;FOLD SLIN P379 Vel=1 m/s CPDAT379 Tool[4]:Microflown3D Base[2]:straight_sol;%{PE}
;FOLD Parameters ;%{h}
;Params IlfProvider=kukaroboter.basistech.inlineforms.movement.spline; Kuka.IsGlobalPoint=False; Kuka.PointName=P379; Kuka.BlendingEnabled=False; Kuka.MoveDataName=CPDAT379; Kuka.VelocityPath=1.000; Kuka.VelocityFieldEnabled=True; Kuka.ColDetectFieldEnabled=True; Kuka.CurrentCDSetIndex=0; Kuka.MovementParameterFieldEnabled=True; IlfCommand=SLIN
;ENDFOLD
SLIN XP379 WITH $VEL = SVEL_CP(2.0, , LCPDAT379),$TOOL = STOOL2(FP379),$BASE = SBASE(FP379.BASE_NO),$IPO_MODE = SIPO_MODE(FP379.IPO_FRAME),$LOAD = SLOAD(FP379.TOOL_NO),$ACC = SACC_CP(LCPDAT379),$ORI_TYPE = SORI_TYP(LCPDAT379),$APO = SAPO(LCPDAT379),$JERK = SJERK(LCPDAT379),$COLLMON_TOL_PRO[1] = USE_CM_PRO_VALUES(0)
;ENDFOLD

;FOLD SLIN P380 Vel=1 m/s CPDAT380 Tool[4]:Microflown3D Base[2]:straight_sol;%{PE}
;FOLD Parameters ;%{h}
;Params IlfProvider=kukaroboter.basistech.inlineforms.movement.spline; Kuka.IsGlobalPoint=False; Kuka.PointName=P380; Kuka.BlendingEnabled=False; Kuka.MoveDataName=CPDAT380; Kuka.VelocityPath=1.000; Kuka.VelocityFieldEnabled=True; Kuka.ColDetectFieldEnabled=True; Kuka.CurrentCDSetIndex=0; Kuka.MovementParameterFieldEnabled=True; IlfCommand=SLIN
;ENDFOLD
SLIN XP380 WITH $VEL = SVEL_CP(2.0, , LCPDAT380),$TOOL = STOOL2(FP380),$BASE = SBASE(FP380.BASE_NO),$IPO_MODE = SIPO_MODE(FP380.IPO_FRAME),$LOAD = SLOAD(FP380.TOOL_NO),$ACC = SACC_CP(LCPDAT380),$ORI_TYPE = SORI_TYP(LCPDAT380),$APO = SAPO(LCPDAT380),$JERK = SJERK(LCPDAT380),$COLLMON_TOL_PRO[1] = USE_CM_PRO_VALUES(0)
;ENDFOLD

;FOLD SLIN P381 Vel=1 m/s CPDAT381 Tool[4]:Microflown3D Base[2]:straight_sol;%{PE}
;FOLD Parameters ;%{h}
;Params IlfProvider=kukaroboter.basistech.inlineforms.movement.spline; Kuka.IsGlobalPoint=False; Kuka.PointName=P381; Kuka.BlendingEnabled=False; Kuka.MoveDataName=CPDAT381; Kuka.VelocityPath=1.000; Kuka.VelocityFieldEnabled=True; Kuka.ColDetectFieldEnabled=True; Kuka.CurrentCDSetIndex=0; Kuka.MovementParameterFieldEnabled=True; IlfCommand=SLIN
;ENDFOLD
SLIN XP381 WITH $VEL = SVEL_CP(2.0, , LCPDAT381),$TOOL = STOOL2(FP381),$BASE = SBASE(FP381.BASE_NO),$IPO_MODE = SIPO_MODE(FP381.IPO_FRAME),$LOAD = SLOAD(FP381.TOOL_NO),$ACC = SACC_CP(LCPDAT381),$ORI_TYPE = SORI_TYP(LCPDAT381),$APO = SAPO(LCPDAT381),$JERK = SJERK(LCPDAT381),$COLLMON_TOL_PRO[1] = USE_CM_PRO_VALUES(0)
;ENDFOLD

;FOLD SLIN P382 Vel=1 m/s CPDAT382 Tool[4]:Microflown3D Base[2]:straight_sol;%{PE}
;FOLD Parameters ;%{h}
;Params IlfProvider=kukaroboter.basistech.inlineforms.movement.spline; Kuka.IsGlobalPoint=False; Kuka.PointName=P382; Kuka.BlendingEnabled=False; Kuka.MoveDataName=CPDAT382; Kuka.VelocityPath=1.000; Kuka.VelocityFieldEnabled=True; Kuka.ColDetectFieldEnabled=True; Kuka.CurrentCDSetIndex=0; Kuka.MovementParameterFieldEnabled=True; IlfCommand=SLIN
;ENDFOLD
SLIN XP382 WITH $VEL = SVEL_CP(2.0, , LCPDAT382),$TOOL = STOOL2(FP382),$BASE = SBASE(FP382.BASE_NO),$IPO_MODE = SIPO_MODE(FP382.IPO_FRAME),$LOAD = SLOAD(FP382.TOOL_NO),$ACC = SACC_CP(LCPDAT382),$ORI_TYPE = SORI_TYP(LCPDAT382),$APO = SAPO(LCPDAT382),$JERK = SJERK(LCPDAT382),$COLLMON_TOL_PRO[1] = USE_CM_PRO_VALUES(0)
;ENDFOLD

;FOLD SLIN P383 Vel=1 m/s CPDAT383 Tool[4]:Microflown3D Base[2]:straight_sol;%{PE}
;FOLD Parameters ;%{h}
;Params IlfProvider=kukaroboter.basistech.inlineforms.movement.spline; Kuka.IsGlobalPoint=False; Kuka.PointName=P383; Kuka.BlendingEnabled=False; Kuka.MoveDataName=CPDAT383; Kuka.VelocityPath=1.000; Kuka.VelocityFieldEnabled=True; Kuka.ColDetectFieldEnabled=True; Kuka.CurrentCDSetIndex=0; Kuka.MovementParameterFieldEnabled=True; IlfCommand=SLIN
;ENDFOLD
SLIN XP383 WITH $VEL = SVEL_CP(2.0, , LCPDAT383),$TOOL = STOOL2(FP383),$BASE = SBASE(FP383.BASE_NO),$IPO_MODE = SIPO_MODE(FP383.IPO_FRAME),$LOAD = SLOAD(FP383.TOOL_NO),$ACC = SACC_CP(LCPDAT383),$ORI_TYPE = SORI_TYP(LCPDAT383),$APO = SAPO(LCPDAT383),$JERK = SJERK(LCPDAT383),$COLLMON_TOL_PRO[1] = USE_CM_PRO_VALUES(0)
;ENDFOLD

;FOLD SLIN P384 Vel=1 m/s CPDAT384 Tool[4]:Microflown3D Base[2]:straight_sol;%{PE}
;FOLD Parameters ;%{h}
;Params IlfProvider=kukaroboter.basistech.inlineforms.movement.spline; Kuka.IsGlobalPoint=False; Kuka.PointName=P384; Kuka.BlendingEnabled=False; Kuka.MoveDataName=CPDAT384; Kuka.VelocityPath=1.000; Kuka.VelocityFieldEnabled=True; Kuka.ColDetectFieldEnabled=True; Kuka.CurrentCDSetIndex=0; Kuka.MovementParameterFieldEnabled=True; IlfCommand=SLIN
;ENDFOLD
SLIN XP384 WITH $VEL = SVEL_CP(2.0, , LCPDAT384),$TOOL = STOOL2(FP384),$BASE = SBASE(FP384.BASE_NO),$IPO_MODE = SIPO_MODE(FP384.IPO_FRAME),$LOAD = SLOAD(FP384.TOOL_NO),$ACC = SACC_CP(LCPDAT384),$ORI_TYPE = SORI_TYP(LCPDAT384),$APO = SAPO(LCPDAT384),$JERK = SJERK(LCPDAT384),$COLLMON_TOL_PRO[1] = USE_CM_PRO_VALUES(0)
;ENDFOLD

;FOLD SLIN P385 Vel=1 m/s CPDAT385 Tool[4]:Microflown3D Base[2]:straight_sol;%{PE}
;FOLD Parameters ;%{h}
;Params IlfProvider=kukaroboter.basistech.inlineforms.movement.spline; Kuka.IsGlobalPoint=False; Kuka.PointName=P385; Kuka.BlendingEnabled=False; Kuka.MoveDataName=CPDAT385; Kuka.VelocityPath=1.000; Kuka.VelocityFieldEnabled=True; Kuka.ColDetectFieldEnabled=True; Kuka.CurrentCDSetIndex=0; Kuka.MovementParameterFieldEnabled=True; IlfCommand=SLIN
;ENDFOLD
SLIN XP385 WITH $VEL = SVEL_CP(2.0, , LCPDAT385),$TOOL = STOOL2(FP385),$BASE = SBASE(FP385.BASE_NO),$IPO_MODE = SIPO_MODE(FP385.IPO_FRAME),$LOAD = SLOAD(FP385.TOOL_NO),$ACC = SACC_CP(LCPDAT385),$ORI_TYPE = SORI_TYP(LCPDAT385),$APO = SAPO(LCPDAT385),$JERK = SJERK(LCPDAT385),$COLLMON_TOL_PRO[1] = USE_CM_PRO_VALUES(0)
;ENDFOLD

;FOLD SLIN P386 Vel=1 m/s CPDAT386 Tool[4]:Microflown3D Base[2]:straight_sol;%{PE}
;FOLD Parameters ;%{h}
;Params IlfProvider=kukaroboter.basistech.inlineforms.movement.spline; Kuka.IsGlobalPoint=False; Kuka.PointName=P386; Kuka.BlendingEnabled=False; Kuka.MoveDataName=CPDAT386; Kuka.VelocityPath=1.000; Kuka.VelocityFieldEnabled=True; Kuka.ColDetectFieldEnabled=True; Kuka.CurrentCDSetIndex=0; Kuka.MovementParameterFieldEnabled=True; IlfCommand=SLIN
;ENDFOLD
SLIN XP386 WITH $VEL = SVEL_CP(2.0, , LCPDAT386),$TOOL = STOOL2(FP386),$BASE = SBASE(FP386.BASE_NO),$IPO_MODE = SIPO_MODE(FP386.IPO_FRAME),$LOAD = SLOAD(FP386.TOOL_NO),$ACC = SACC_CP(LCPDAT386),$ORI_TYPE = SORI_TYP(LCPDAT386),$APO = SAPO(LCPDAT386),$JERK = SJERK(LCPDAT386),$COLLMON_TOL_PRO[1] = USE_CM_PRO_VALUES(0)
;ENDFOLD

;FOLD SLIN P387 Vel=1 m/s CPDAT387 Tool[4]:Microflown3D Base[2]:straight_sol;%{PE}
;FOLD Parameters ;%{h}
;Params IlfProvider=kukaroboter.basistech.inlineforms.movement.spline; Kuka.IsGlobalPoint=False; Kuka.PointName=P387; Kuka.BlendingEnabled=False; Kuka.MoveDataName=CPDAT387; Kuka.VelocityPath=1.000; Kuka.VelocityFieldEnabled=True; Kuka.ColDetectFieldEnabled=True; Kuka.CurrentCDSetIndex=0; Kuka.MovementParameterFieldEnabled=True; IlfCommand=SLIN
;ENDFOLD
SLIN XP387 WITH $VEL = SVEL_CP(2.0, , LCPDAT387),$TOOL = STOOL2(FP387),$BASE = SBASE(FP387.BASE_NO),$IPO_MODE = SIPO_MODE(FP387.IPO_FRAME),$LOAD = SLOAD(FP387.TOOL_NO),$ACC = SACC_CP(LCPDAT387),$ORI_TYPE = SORI_TYP(LCPDAT387),$APO = SAPO(LCPDAT387),$JERK = SJERK(LCPDAT387),$COLLMON_TOL_PRO[1] = USE_CM_PRO_VALUES(0)
;ENDFOLD

;FOLD SLIN P388 Vel=1 m/s CPDAT388 Tool[4]:Microflown3D Base[2]:straight_sol;%{PE}
;FOLD Parameters ;%{h}
;Params IlfProvider=kukaroboter.basistech.inlineforms.movement.spline; Kuka.IsGlobalPoint=False; Kuka.PointName=P388; Kuka.BlendingEnabled=False; Kuka.MoveDataName=CPDAT388; Kuka.VelocityPath=1.000; Kuka.VelocityFieldEnabled=True; Kuka.ColDetectFieldEnabled=True; Kuka.CurrentCDSetIndex=0; Kuka.MovementParameterFieldEnabled=True; IlfCommand=SLIN
;ENDFOLD
SLIN XP388 WITH $VEL = SVEL_CP(2.0, , LCPDAT388),$TOOL = STOOL2(FP388),$BASE = SBASE(FP388.BASE_NO),$IPO_MODE = SIPO_MODE(FP388.IPO_FRAME),$LOAD = SLOAD(FP388.TOOL_NO),$ACC = SACC_CP(LCPDAT388),$ORI_TYPE = SORI_TYP(LCPDAT388),$APO = SAPO(LCPDAT388),$JERK = SJERK(LCPDAT388),$COLLMON_TOL_PRO[1] = USE_CM_PRO_VALUES(0)
;ENDFOLD

;FOLD SLIN P389 Vel=1 m/s CPDAT389 Tool[4]:Microflown3D Base[2]:straight_sol;%{PE}
;FOLD Parameters ;%{h}
;Params IlfProvider=kukaroboter.basistech.inlineforms.movement.spline; Kuka.IsGlobalPoint=False; Kuka.PointName=P389; Kuka.BlendingEnabled=False; Kuka.MoveDataName=CPDAT389; Kuka.VelocityPath=1.000; Kuka.VelocityFieldEnabled=True; Kuka.ColDetectFieldEnabled=True; Kuka.CurrentCDSetIndex=0; Kuka.MovementParameterFieldEnabled=True; IlfCommand=SLIN
;ENDFOLD
SLIN XP389 WITH $VEL = SVEL_CP(2.0, , LCPDAT389),$TOOL = STOOL2(FP389),$BASE = SBASE(FP389.BASE_NO),$IPO_MODE = SIPO_MODE(FP389.IPO_FRAME),$LOAD = SLOAD(FP389.TOOL_NO),$ACC = SACC_CP(LCPDAT389),$ORI_TYPE = SORI_TYP(LCPDAT389),$APO = SAPO(LCPDAT389),$JERK = SJERK(LCPDAT389),$COLLMON_TOL_PRO[1] = USE_CM_PRO_VALUES(0)
;ENDFOLD

;FOLD SLIN P390 Vel=1 m/s CPDAT390 Tool[4]:Microflown3D Base[2]:straight_sol;%{PE}
;FOLD Parameters ;%{h}
;Params IlfProvider=kukaroboter.basistech.inlineforms.movement.spline; Kuka.IsGlobalPoint=False; Kuka.PointName=P390; Kuka.BlendingEnabled=False; Kuka.MoveDataName=CPDAT390; Kuka.VelocityPath=1.000; Kuka.VelocityFieldEnabled=True; Kuka.ColDetectFieldEnabled=True; Kuka.CurrentCDSetIndex=0; Kuka.MovementParameterFieldEnabled=True; IlfCommand=SLIN
;ENDFOLD
SLIN XP390 WITH $VEL = SVEL_CP(2.0, , LCPDAT390),$TOOL = STOOL2(FP390),$BASE = SBASE(FP390.BASE_NO),$IPO_MODE = SIPO_MODE(FP390.IPO_FRAME),$LOAD = SLOAD(FP390.TOOL_NO),$ACC = SACC_CP(LCPDAT390),$ORI_TYPE = SORI_TYP(LCPDAT390),$APO = SAPO(LCPDAT390),$JERK = SJERK(LCPDAT390),$COLLMON_TOL_PRO[1] = USE_CM_PRO_VALUES(0)
;ENDFOLD

;FOLD SLIN P391 Vel=1 m/s CPDAT391 Tool[4]:Microflown3D Base[2]:straight_sol;%{PE}
;FOLD Parameters ;%{h}
;Params IlfProvider=kukaroboter.basistech.inlineforms.movement.spline; Kuka.IsGlobalPoint=False; Kuka.PointName=P391; Kuka.BlendingEnabled=False; Kuka.MoveDataName=CPDAT391; Kuka.VelocityPath=1.000; Kuka.VelocityFieldEnabled=True; Kuka.ColDetectFieldEnabled=True; Kuka.CurrentCDSetIndex=0; Kuka.MovementParameterFieldEnabled=True; IlfCommand=SLIN
;ENDFOLD
SLIN XP391 WITH $VEL = SVEL_CP(2.0, , LCPDAT391),$TOOL = STOOL2(FP391),$BASE = SBASE(FP391.BASE_NO),$IPO_MODE = SIPO_MODE(FP391.IPO_FRAME),$LOAD = SLOAD(FP391.TOOL_NO),$ACC = SACC_CP(LCPDAT391),$ORI_TYPE = SORI_TYP(LCPDAT391),$APO = SAPO(LCPDAT391),$JERK = SJERK(LCPDAT391),$COLLMON_TOL_PRO[1] = USE_CM_PRO_VALUES(0)
;ENDFOLD

;FOLD SLIN P392 Vel=1 m/s CPDAT392 Tool[4]:Microflown3D Base[2]:straight_sol;%{PE}
;FOLD Parameters ;%{h}
;Params IlfProvider=kukaroboter.basistech.inlineforms.movement.spline; Kuka.IsGlobalPoint=False; Kuka.PointName=P392; Kuka.BlendingEnabled=False; Kuka.MoveDataName=CPDAT392; Kuka.VelocityPath=1.000; Kuka.VelocityFieldEnabled=True; Kuka.ColDetectFieldEnabled=True; Kuka.CurrentCDSetIndex=0; Kuka.MovementParameterFieldEnabled=True; IlfCommand=SLIN
;ENDFOLD
SLIN XP392 WITH $VEL = SVEL_CP(2.0, , LCPDAT392),$TOOL = STOOL2(FP392),$BASE = SBASE(FP392.BASE_NO),$IPO_MODE = SIPO_MODE(FP392.IPO_FRAME),$LOAD = SLOAD(FP392.TOOL_NO),$ACC = SACC_CP(LCPDAT392),$ORI_TYPE = SORI_TYP(LCPDAT392),$APO = SAPO(LCPDAT392),$JERK = SJERK(LCPDAT392),$COLLMON_TOL_PRO[1] = USE_CM_PRO_VALUES(0)
;ENDFOLD

;FOLD SLIN P393 Vel=1 m/s CPDAT393 Tool[4]:Microflown3D Base[2]:straight_sol;%{PE}
;FOLD Parameters ;%{h}
;Params IlfProvider=kukaroboter.basistech.inlineforms.movement.spline; Kuka.IsGlobalPoint=False; Kuka.PointName=P393; Kuka.BlendingEnabled=False; Kuka.MoveDataName=CPDAT393; Kuka.VelocityPath=1.000; Kuka.VelocityFieldEnabled=True; Kuka.ColDetectFieldEnabled=True; Kuka.CurrentCDSetIndex=0; Kuka.MovementParameterFieldEnabled=True; IlfCommand=SLIN
;ENDFOLD
SLIN XP393 WITH $VEL = SVEL_CP(2.0, , LCPDAT393),$TOOL = STOOL2(FP393),$BASE = SBASE(FP393.BASE_NO),$IPO_MODE = SIPO_MODE(FP393.IPO_FRAME),$LOAD = SLOAD(FP393.TOOL_NO),$ACC = SACC_CP(LCPDAT393),$ORI_TYPE = SORI_TYP(LCPDAT393),$APO = SAPO(LCPDAT393),$JERK = SJERK(LCPDAT393),$COLLMON_TOL_PRO[1] = USE_CM_PRO_VALUES(0)
;ENDFOLD

;FOLD SLIN P394 Vel=1 m/s CPDAT394 Tool[4]:Microflown3D Base[2]:straight_sol;%{PE}
;FOLD Parameters ;%{h}
;Params IlfProvider=kukaroboter.basistech.inlineforms.movement.spline; Kuka.IsGlobalPoint=False; Kuka.PointName=P394; Kuka.BlendingEnabled=False; Kuka.MoveDataName=CPDAT394; Kuka.VelocityPath=1.000; Kuka.VelocityFieldEnabled=True; Kuka.ColDetectFieldEnabled=True; Kuka.CurrentCDSetIndex=0; Kuka.MovementParameterFieldEnabled=True; IlfCommand=SLIN
;ENDFOLD
SLIN XP394 WITH $VEL = SVEL_CP(2.0, , LCPDAT394),$TOOL = STOOL2(FP394),$BASE = SBASE(FP394.BASE_NO),$IPO_MODE = SIPO_MODE(FP394.IPO_FRAME),$LOAD = SLOAD(FP394.TOOL_NO),$ACC = SACC_CP(LCPDAT394),$ORI_TYPE = SORI_TYP(LCPDAT394),$APO = SAPO(LCPDAT394),$JERK = SJERK(LCPDAT394),$COLLMON_TOL_PRO[1] = USE_CM_PRO_VALUES(0)
;ENDFOLD

;FOLD SLIN P395 Vel=1 m/s CPDAT395 Tool[4]:Microflown3D Base[2]:straight_sol;%{PE}
;FOLD Parameters ;%{h}
;Params IlfProvider=kukaroboter.basistech.inlineforms.movement.spline; Kuka.IsGlobalPoint=False; Kuka.PointName=P395; Kuka.BlendingEnabled=False; Kuka.MoveDataName=CPDAT395; Kuka.VelocityPath=1.000; Kuka.VelocityFieldEnabled=True; Kuka.ColDetectFieldEnabled=True; Kuka.CurrentCDSetIndex=0; Kuka.MovementParameterFieldEnabled=True; IlfCommand=SLIN
;ENDFOLD
SLIN XP395 WITH $VEL = SVEL_CP(2.0, , LCPDAT395),$TOOL = STOOL2(FP395),$BASE = SBASE(FP395.BASE_NO),$IPO_MODE = SIPO_MODE(FP395.IPO_FRAME),$LOAD = SLOAD(FP395.TOOL_NO),$ACC = SACC_CP(LCPDAT395),$ORI_TYPE = SORI_TYP(LCPDAT395),$APO = SAPO(LCPDAT395),$JERK = SJERK(LCPDAT395),$COLLMON_TOL_PRO[1] = USE_CM_PRO_VALUES(0)
;ENDFOLD

;FOLD SLIN P396 Vel=1 m/s CPDAT396 Tool[4]:Microflown3D Base[2]:straight_sol;%{PE}
;FOLD Parameters ;%{h}
;Params IlfProvider=kukaroboter.basistech.inlineforms.movement.spline; Kuka.IsGlobalPoint=False; Kuka.PointName=P396; Kuka.BlendingEnabled=False; Kuka.MoveDataName=CPDAT396; Kuka.VelocityPath=1.000; Kuka.VelocityFieldEnabled=True; Kuka.ColDetectFieldEnabled=True; Kuka.CurrentCDSetIndex=0; Kuka.MovementParameterFieldEnabled=True; IlfCommand=SLIN
;ENDFOLD
SLIN XP396 WITH $VEL = SVEL_CP(2.0, , LCPDAT396),$TOOL = STOOL2(FP396),$BASE = SBASE(FP396.BASE_NO),$IPO_MODE = SIPO_MODE(FP396.IPO_FRAME),$LOAD = SLOAD(FP396.TOOL_NO),$ACC = SACC_CP(LCPDAT396),$ORI_TYPE = SORI_TYP(LCPDAT396),$APO = SAPO(LCPDAT396),$JERK = SJERK(LCPDAT396),$COLLMON_TOL_PRO[1] = USE_CM_PRO_VALUES(0)
;ENDFOLD

;FOLD SLIN P397 Vel=1 m/s CPDAT397 Tool[4]:Microflown3D Base[2]:straight_sol;%{PE}
;FOLD Parameters ;%{h}
;Params IlfProvider=kukaroboter.basistech.inlineforms.movement.spline; Kuka.IsGlobalPoint=False; Kuka.PointName=P397; Kuka.BlendingEnabled=False; Kuka.MoveDataName=CPDAT397; Kuka.VelocityPath=1.000; Kuka.VelocityFieldEnabled=True; Kuka.ColDetectFieldEnabled=True; Kuka.CurrentCDSetIndex=0; Kuka.MovementParameterFieldEnabled=True; IlfCommand=SLIN
;ENDFOLD
SLIN XP397 WITH $VEL = SVEL_CP(2.0, , LCPDAT397),$TOOL = STOOL2(FP397),$BASE = SBASE(FP397.BASE_NO),$IPO_MODE = SIPO_MODE(FP397.IPO_FRAME),$LOAD = SLOAD(FP397.TOOL_NO),$ACC = SACC_CP(LCPDAT397),$ORI_TYPE = SORI_TYP(LCPDAT397),$APO = SAPO(LCPDAT397),$JERK = SJERK(LCPDAT397),$COLLMON_TOL_PRO[1] = USE_CM_PRO_VALUES(0)
;ENDFOLD

;FOLD SLIN P398 Vel=1 m/s CPDAT398 Tool[4]:Microflown3D Base[2]:straight_sol;%{PE}
;FOLD Parameters ;%{h}
;Params IlfProvider=kukaroboter.basistech.inlineforms.movement.spline; Kuka.IsGlobalPoint=False; Kuka.PointName=P398; Kuka.BlendingEnabled=False; Kuka.MoveDataName=CPDAT398; Kuka.VelocityPath=1.000; Kuka.VelocityFieldEnabled=True; Kuka.ColDetectFieldEnabled=True; Kuka.CurrentCDSetIndex=0; Kuka.MovementParameterFieldEnabled=True; IlfCommand=SLIN
;ENDFOLD
SLIN XP398 WITH $VEL = SVEL_CP(2.0, , LCPDAT398),$TOOL = STOOL2(FP398),$BASE = SBASE(FP398.BASE_NO),$IPO_MODE = SIPO_MODE(FP398.IPO_FRAME),$LOAD = SLOAD(FP398.TOOL_NO),$ACC = SACC_CP(LCPDAT398),$ORI_TYPE = SORI_TYP(LCPDAT398),$APO = SAPO(LCPDAT398),$JERK = SJERK(LCPDAT398),$COLLMON_TOL_PRO[1] = USE_CM_PRO_VALUES(0)
;ENDFOLD

;FOLD SLIN P399 Vel=1 m/s CPDAT399 Tool[4]:Microflown3D Base[2]:straight_sol;%{PE}
;FOLD Parameters ;%{h}
;Params IlfProvider=kukaroboter.basistech.inlineforms.movement.spline; Kuka.IsGlobalPoint=False; Kuka.PointName=P399; Kuka.BlendingEnabled=False; Kuka.MoveDataName=CPDAT399; Kuka.VelocityPath=1.000; Kuka.VelocityFieldEnabled=True; Kuka.ColDetectFieldEnabled=True; Kuka.CurrentCDSetIndex=0; Kuka.MovementParameterFieldEnabled=True; IlfCommand=SLIN
;ENDFOLD
SLIN XP399 WITH $VEL = SVEL_CP(2.0, , LCPDAT399),$TOOL = STOOL2(FP399),$BASE = SBASE(FP399.BASE_NO),$IPO_MODE = SIPO_MODE(FP399.IPO_FRAME),$LOAD = SLOAD(FP399.TOOL_NO),$ACC = SACC_CP(LCPDAT399),$ORI_TYPE = SORI_TYP(LCPDAT399),$APO = SAPO(LCPDAT399),$JERK = SJERK(LCPDAT399),$COLLMON_TOL_PRO[1] = USE_CM_PRO_VALUES(0)
;ENDFOLD

;FOLD SLIN P400 Vel=1 m/s CPDAT400 Tool[4]:Microflown3D Base[2]:straight_sol;%{PE}
;FOLD Parameters ;%{h}
;Params IlfProvider=kukaroboter.basistech.inlineforms.movement.spline; Kuka.IsGlobalPoint=False; Kuka.PointName=P400; Kuka.BlendingEnabled=False; Kuka.MoveDataName=CPDAT400; Kuka.VelocityPath=1.000; Kuka.VelocityFieldEnabled=True; Kuka.ColDetectFieldEnabled=True; Kuka.CurrentCDSetIndex=0; Kuka.MovementParameterFieldEnabled=True; IlfCommand=SLIN
;ENDFOLD
SLIN XP400 WITH $VEL = SVEL_CP(2.0, , LCPDAT400),$TOOL = STOOL2(FP400),$BASE = SBASE(FP400.BASE_NO),$IPO_MODE = SIPO_MODE(FP400.IPO_FRAME),$LOAD = SLOAD(FP400.TOOL_NO),$ACC = SACC_CP(LCPDAT400),$ORI_TYPE = SORI_TYP(LCPDAT400),$APO = SAPO(LCPDAT400),$JERK = SJERK(LCPDAT400),$COLLMON_TOL_PRO[1] = USE_CM_PRO_VALUES(0)
;ENDFOLD

;FOLD SLIN P401 Vel=1 m/s CPDAT401 Tool[4]:Microflown3D Base[2]:straight_sol;%{PE}
;FOLD Parameters ;%{h}
;Params IlfProvider=kukaroboter.basistech.inlineforms.movement.spline; Kuka.IsGlobalPoint=False; Kuka.PointName=P401; Kuka.BlendingEnabled=False; Kuka.MoveDataName=CPDAT401; Kuka.VelocityPath=1.000; Kuka.VelocityFieldEnabled=True; Kuka.ColDetectFieldEnabled=True; Kuka.CurrentCDSetIndex=0; Kuka.MovementParameterFieldEnabled=True; IlfCommand=SLIN
;ENDFOLD
SLIN XP401 WITH $VEL = SVEL_CP(2.0, , LCPDAT401),$TOOL = STOOL2(FP401),$BASE = SBASE(FP401.BASE_NO),$IPO_MODE = SIPO_MODE(FP401.IPO_FRAME),$LOAD = SLOAD(FP401.TOOL_NO),$ACC = SACC_CP(LCPDAT401),$ORI_TYPE = SORI_TYP(LCPDAT401),$APO = SAPO(LCPDAT401),$JERK = SJERK(LCPDAT401),$COLLMON_TOL_PRO[1] = USE_CM_PRO_VALUES(0)
;ENDFOLD

;FOLD SLIN P402 Vel=1 m/s CPDAT402 Tool[4]:Microflown3D Base[2]:straight_sol;%{PE}
;FOLD Parameters ;%{h}
;Params IlfProvider=kukaroboter.basistech.inlineforms.movement.spline; Kuka.IsGlobalPoint=False; Kuka.PointName=P402; Kuka.BlendingEnabled=False; Kuka.MoveDataName=CPDAT402; Kuka.VelocityPath=1.000; Kuka.VelocityFieldEnabled=True; Kuka.ColDetectFieldEnabled=True; Kuka.CurrentCDSetIndex=0; Kuka.MovementParameterFieldEnabled=True; IlfCommand=SLIN
;ENDFOLD
SLIN XP402 WITH $VEL = SVEL_CP(2.0, , LCPDAT402),$TOOL = STOOL2(FP402),$BASE = SBASE(FP402.BASE_NO),$IPO_MODE = SIPO_MODE(FP402.IPO_FRAME),$LOAD = SLOAD(FP402.TOOL_NO),$ACC = SACC_CP(LCPDAT402),$ORI_TYPE = SORI_TYP(LCPDAT402),$APO = SAPO(LCPDAT402),$JERK = SJERK(LCPDAT402),$COLLMON_TOL_PRO[1] = USE_CM_PRO_VALUES(0)
;ENDFOLD

;FOLD SLIN P403 Vel=1 m/s CPDAT403 Tool[4]:Microflown3D Base[2]:straight_sol;%{PE}
;FOLD Parameters ;%{h}
;Params IlfProvider=kukaroboter.basistech.inlineforms.movement.spline; Kuka.IsGlobalPoint=False; Kuka.PointName=P403; Kuka.BlendingEnabled=False; Kuka.MoveDataName=CPDAT403; Kuka.VelocityPath=1.000; Kuka.VelocityFieldEnabled=True; Kuka.ColDetectFieldEnabled=True; Kuka.CurrentCDSetIndex=0; Kuka.MovementParameterFieldEnabled=True; IlfCommand=SLIN
;ENDFOLD
SLIN XP403 WITH $VEL = SVEL_CP(2.0, , LCPDAT403),$TOOL = STOOL2(FP403),$BASE = SBASE(FP403.BASE_NO),$IPO_MODE = SIPO_MODE(FP403.IPO_FRAME),$LOAD = SLOAD(FP403.TOOL_NO),$ACC = SACC_CP(LCPDAT403),$ORI_TYPE = SORI_TYP(LCPDAT403),$APO = SAPO(LCPDAT403),$JERK = SJERK(LCPDAT403),$COLLMON_TOL_PRO[1] = USE_CM_PRO_VALUES(0)
;ENDFOLD

;FOLD SLIN P404 Vel=1 m/s CPDAT404 Tool[4]:Microflown3D Base[2]:straight_sol;%{PE}
;FOLD Parameters ;%{h}
;Params IlfProvider=kukaroboter.basistech.inlineforms.movement.spline; Kuka.IsGlobalPoint=False; Kuka.PointName=P404; Kuka.BlendingEnabled=False; Kuka.MoveDataName=CPDAT404; Kuka.VelocityPath=1.000; Kuka.VelocityFieldEnabled=True; Kuka.ColDetectFieldEnabled=True; Kuka.CurrentCDSetIndex=0; Kuka.MovementParameterFieldEnabled=True; IlfCommand=SLIN
;ENDFOLD
SLIN XP404 WITH $VEL = SVEL_CP(2.0, , LCPDAT404),$TOOL = STOOL2(FP404),$BASE = SBASE(FP404.BASE_NO),$IPO_MODE = SIPO_MODE(FP404.IPO_FRAME),$LOAD = SLOAD(FP404.TOOL_NO),$ACC = SACC_CP(LCPDAT404),$ORI_TYPE = SORI_TYP(LCPDAT404),$APO = SAPO(LCPDAT404),$JERK = SJERK(LCPDAT404),$COLLMON_TOL_PRO[1] = USE_CM_PRO_VALUES(0)
;ENDFOLD

;FOLD SLIN P405 Vel=1 m/s CPDAT405 Tool[4]:Microflown3D Base[2]:straight_sol;%{PE}
;FOLD Parameters ;%{h}
;Params IlfProvider=kukaroboter.basistech.inlineforms.movement.spline; Kuka.IsGlobalPoint=False; Kuka.PointName=P405; Kuka.BlendingEnabled=False; Kuka.MoveDataName=CPDAT405; Kuka.VelocityPath=1.000; Kuka.VelocityFieldEnabled=True; Kuka.ColDetectFieldEnabled=True; Kuka.CurrentCDSetIndex=0; Kuka.MovementParameterFieldEnabled=True; IlfCommand=SLIN
;ENDFOLD
SLIN XP405 WITH $VEL = SVEL_CP(2.0, , LCPDAT405),$TOOL = STOOL2(FP405),$BASE = SBASE(FP405.BASE_NO),$IPO_MODE = SIPO_MODE(FP405.IPO_FRAME),$LOAD = SLOAD(FP405.TOOL_NO),$ACC = SACC_CP(LCPDAT405),$ORI_TYPE = SORI_TYP(LCPDAT405),$APO = SAPO(LCPDAT405),$JERK = SJERK(LCPDAT405),$COLLMON_TOL_PRO[1] = USE_CM_PRO_VALUES(0)
;ENDFOLD

;FOLD SLIN P406 Vel=1 m/s CPDAT406 Tool[4]:Microflown3D Base[2]:straight_sol;%{PE}
;FOLD Parameters ;%{h}
;Params IlfProvider=kukaroboter.basistech.inlineforms.movement.spline; Kuka.IsGlobalPoint=False; Kuka.PointName=P406; Kuka.BlendingEnabled=False; Kuka.MoveDataName=CPDAT406; Kuka.VelocityPath=1.000; Kuka.VelocityFieldEnabled=True; Kuka.ColDetectFieldEnabled=True; Kuka.CurrentCDSetIndex=0; Kuka.MovementParameterFieldEnabled=True; IlfCommand=SLIN
;ENDFOLD
SLIN XP406 WITH $VEL = SVEL_CP(2.0, , LCPDAT406),$TOOL = STOOL2(FP406),$BASE = SBASE(FP406.BASE_NO),$IPO_MODE = SIPO_MODE(FP406.IPO_FRAME),$LOAD = SLOAD(FP406.TOOL_NO),$ACC = SACC_CP(LCPDAT406),$ORI_TYPE = SORI_TYP(LCPDAT406),$APO = SAPO(LCPDAT406),$JERK = SJERK(LCPDAT406),$COLLMON_TOL_PRO[1] = USE_CM_PRO_VALUES(0)
;ENDFOLD

;FOLD SLIN P407 Vel=1 m/s CPDAT407 Tool[4]:Microflown3D Base[2]:straight_sol;%{PE}
;FOLD Parameters ;%{h}
;Params IlfProvider=kukaroboter.basistech.inlineforms.movement.spline; Kuka.IsGlobalPoint=False; Kuka.PointName=P407; Kuka.BlendingEnabled=False; Kuka.MoveDataName=CPDAT407; Kuka.VelocityPath=1.000; Kuka.VelocityFieldEnabled=True; Kuka.ColDetectFieldEnabled=True; Kuka.CurrentCDSetIndex=0; Kuka.MovementParameterFieldEnabled=True; IlfCommand=SLIN
;ENDFOLD
SLIN XP407 WITH $VEL = SVEL_CP(2.0, , LCPDAT407),$TOOL = STOOL2(FP407),$BASE = SBASE(FP407.BASE_NO),$IPO_MODE = SIPO_MODE(FP407.IPO_FRAME),$LOAD = SLOAD(FP407.TOOL_NO),$ACC = SACC_CP(LCPDAT407),$ORI_TYPE = SORI_TYP(LCPDAT407),$APO = SAPO(LCPDAT407),$JERK = SJERK(LCPDAT407),$COLLMON_TOL_PRO[1] = USE_CM_PRO_VALUES(0)
;ENDFOLD

;FOLD SLIN P408 Vel=1 m/s CPDAT408 Tool[4]:Microflown3D Base[2]:straight_sol;%{PE}
;FOLD Parameters ;%{h}
;Params IlfProvider=kukaroboter.basistech.inlineforms.movement.spline; Kuka.IsGlobalPoint=False; Kuka.PointName=P408; Kuka.BlendingEnabled=False; Kuka.MoveDataName=CPDAT408; Kuka.VelocityPath=1.000; Kuka.VelocityFieldEnabled=True; Kuka.ColDetectFieldEnabled=True; Kuka.CurrentCDSetIndex=0; Kuka.MovementParameterFieldEnabled=True; IlfCommand=SLIN
;ENDFOLD
SLIN XP408 WITH $VEL = SVEL_CP(2.0, , LCPDAT408),$TOOL = STOOL2(FP408),$BASE = SBASE(FP408.BASE_NO),$IPO_MODE = SIPO_MODE(FP408.IPO_FRAME),$LOAD = SLOAD(FP408.TOOL_NO),$ACC = SACC_CP(LCPDAT408),$ORI_TYPE = SORI_TYP(LCPDAT408),$APO = SAPO(LCPDAT408),$JERK = SJERK(LCPDAT408),$COLLMON_TOL_PRO[1] = USE_CM_PRO_VALUES(0)
;ENDFOLD

;FOLD SLIN P409 Vel=1 m/s CPDAT409 Tool[4]:Microflown3D Base[2]:straight_sol;%{PE}
;FOLD Parameters ;%{h}
;Params IlfProvider=kukaroboter.basistech.inlineforms.movement.spline; Kuka.IsGlobalPoint=False; Kuka.PointName=P409; Kuka.BlendingEnabled=False; Kuka.MoveDataName=CPDAT409; Kuka.VelocityPath=1.000; Kuka.VelocityFieldEnabled=True; Kuka.ColDetectFieldEnabled=True; Kuka.CurrentCDSetIndex=0; Kuka.MovementParameterFieldEnabled=True; IlfCommand=SLIN
;ENDFOLD
SLIN XP409 WITH $VEL = SVEL_CP(2.0, , LCPDAT409),$TOOL = STOOL2(FP409),$BASE = SBASE(FP409.BASE_NO),$IPO_MODE = SIPO_MODE(FP409.IPO_FRAME),$LOAD = SLOAD(FP409.TOOL_NO),$ACC = SACC_CP(LCPDAT409),$ORI_TYPE = SORI_TYP(LCPDAT409),$APO = SAPO(LCPDAT409),$JERK = SJERK(LCPDAT409),$COLLMON_TOL_PRO[1] = USE_CM_PRO_VALUES(0)
;ENDFOLD

;FOLD SLIN P410 Vel=1 m/s CPDAT410 Tool[4]:Microflown3D Base[2]:straight_sol;%{PE}
;FOLD Parameters ;%{h}
;Params IlfProvider=kukaroboter.basistech.inlineforms.movement.spline; Kuka.IsGlobalPoint=False; Kuka.PointName=P410; Kuka.BlendingEnabled=False; Kuka.MoveDataName=CPDAT410; Kuka.VelocityPath=1.000; Kuka.VelocityFieldEnabled=True; Kuka.ColDetectFieldEnabled=True; Kuka.CurrentCDSetIndex=0; Kuka.MovementParameterFieldEnabled=True; IlfCommand=SLIN
;ENDFOLD
SLIN XP410 WITH $VEL = SVEL_CP(2.0, , LCPDAT410),$TOOL = STOOL2(FP410),$BASE = SBASE(FP410.BASE_NO),$IPO_MODE = SIPO_MODE(FP410.IPO_FRAME),$LOAD = SLOAD(FP410.TOOL_NO),$ACC = SACC_CP(LCPDAT410),$ORI_TYPE = SORI_TYP(LCPDAT410),$APO = SAPO(LCPDAT410),$JERK = SJERK(LCPDAT410),$COLLMON_TOL_PRO[1] = USE_CM_PRO_VALUES(0)
;ENDFOLD

;FOLD SLIN P411 Vel=1 m/s CPDAT411 Tool[4]:Microflown3D Base[2]:straight_sol;%{PE}
;FOLD Parameters ;%{h}
;Params IlfProvider=kukaroboter.basistech.inlineforms.movement.spline; Kuka.IsGlobalPoint=False; Kuka.PointName=P411; Kuka.BlendingEnabled=False; Kuka.MoveDataName=CPDAT411; Kuka.VelocityPath=1.000; Kuka.VelocityFieldEnabled=True; Kuka.ColDetectFieldEnabled=True; Kuka.CurrentCDSetIndex=0; Kuka.MovementParameterFieldEnabled=True; IlfCommand=SLIN
;ENDFOLD
SLIN XP411 WITH $VEL = SVEL_CP(2.0, , LCPDAT411),$TOOL = STOOL2(FP411),$BASE = SBASE(FP411.BASE_NO),$IPO_MODE = SIPO_MODE(FP411.IPO_FRAME),$LOAD = SLOAD(FP411.TOOL_NO),$ACC = SACC_CP(LCPDAT411),$ORI_TYPE = SORI_TYP(LCPDAT411),$APO = SAPO(LCPDAT411),$JERK = SJERK(LCPDAT411),$COLLMON_TOL_PRO[1] = USE_CM_PRO_VALUES(0)
;ENDFOLD

;FOLD SLIN P412 Vel=1 m/s CPDAT412 Tool[4]:Microflown3D Base[2]:straight_sol;%{PE}
;FOLD Parameters ;%{h}
;Params IlfProvider=kukaroboter.basistech.inlineforms.movement.spline; Kuka.IsGlobalPoint=False; Kuka.PointName=P412; Kuka.BlendingEnabled=False; Kuka.MoveDataName=CPDAT412; Kuka.VelocityPath=1.000; Kuka.VelocityFieldEnabled=True; Kuka.ColDetectFieldEnabled=True; Kuka.CurrentCDSetIndex=0; Kuka.MovementParameterFieldEnabled=True; IlfCommand=SLIN
;ENDFOLD
SLIN XP412 WITH $VEL = SVEL_CP(2.0, , LCPDAT412),$TOOL = STOOL2(FP412),$BASE = SBASE(FP412.BASE_NO),$IPO_MODE = SIPO_MODE(FP412.IPO_FRAME),$LOAD = SLOAD(FP412.TOOL_NO),$ACC = SACC_CP(LCPDAT412),$ORI_TYPE = SORI_TYP(LCPDAT412),$APO = SAPO(LCPDAT412),$JERK = SJERK(LCPDAT412),$COLLMON_TOL_PRO[1] = USE_CM_PRO_VALUES(0)
;ENDFOLD

;FOLD SLIN P413 Vel=1 m/s CPDAT413 Tool[4]:Microflown3D Base[2]:straight_sol;%{PE}
;FOLD Parameters ;%{h}
;Params IlfProvider=kukaroboter.basistech.inlineforms.movement.spline; Kuka.IsGlobalPoint=False; Kuka.PointName=P413; Kuka.BlendingEnabled=False; Kuka.MoveDataName=CPDAT413; Kuka.VelocityPath=1.000; Kuka.VelocityFieldEnabled=True; Kuka.ColDetectFieldEnabled=True; Kuka.CurrentCDSetIndex=0; Kuka.MovementParameterFieldEnabled=True; IlfCommand=SLIN
;ENDFOLD
SLIN XP413 WITH $VEL = SVEL_CP(2.0, , LCPDAT413),$TOOL = STOOL2(FP413),$BASE = SBASE(FP413.BASE_NO),$IPO_MODE = SIPO_MODE(FP413.IPO_FRAME),$LOAD = SLOAD(FP413.TOOL_NO),$ACC = SACC_CP(LCPDAT413),$ORI_TYPE = SORI_TYP(LCPDAT413),$APO = SAPO(LCPDAT413),$JERK = SJERK(LCPDAT413),$COLLMON_TOL_PRO[1] = USE_CM_PRO_VALUES(0)
;ENDFOLD

;FOLD SLIN P414 Vel=1 m/s CPDAT414 Tool[4]:Microflown3D Base[2]:straight_sol;%{PE}
;FOLD Parameters ;%{h}
;Params IlfProvider=kukaroboter.basistech.inlineforms.movement.spline; Kuka.IsGlobalPoint=False; Kuka.PointName=P414; Kuka.BlendingEnabled=False; Kuka.MoveDataName=CPDAT414; Kuka.VelocityPath=1.000; Kuka.VelocityFieldEnabled=True; Kuka.ColDetectFieldEnabled=True; Kuka.CurrentCDSetIndex=0; Kuka.MovementParameterFieldEnabled=True; IlfCommand=SLIN
;ENDFOLD
SLIN XP414 WITH $VEL = SVEL_CP(2.0, , LCPDAT414),$TOOL = STOOL2(FP414),$BASE = SBASE(FP414.BASE_NO),$IPO_MODE = SIPO_MODE(FP414.IPO_FRAME),$LOAD = SLOAD(FP414.TOOL_NO),$ACC = SACC_CP(LCPDAT414),$ORI_TYPE = SORI_TYP(LCPDAT414),$APO = SAPO(LCPDAT414),$JERK = SJERK(LCPDAT414),$COLLMON_TOL_PRO[1] = USE_CM_PRO_VALUES(0)
;ENDFOLD

;FOLD SLIN P415 Vel=1 m/s CPDAT415 Tool[4]:Microflown3D Base[2]:straight_sol;%{PE}
;FOLD Parameters ;%{h}
;Params IlfProvider=kukaroboter.basistech.inlineforms.movement.spline; Kuka.IsGlobalPoint=False; Kuka.PointName=P415; Kuka.BlendingEnabled=False; Kuka.MoveDataName=CPDAT415; Kuka.VelocityPath=1.000; Kuka.VelocityFieldEnabled=True; Kuka.ColDetectFieldEnabled=True; Kuka.CurrentCDSetIndex=0; Kuka.MovementParameterFieldEnabled=True; IlfCommand=SLIN
;ENDFOLD
SLIN XP415 WITH $VEL = SVEL_CP(2.0, , LCPDAT415),$TOOL = STOOL2(FP415),$BASE = SBASE(FP415.BASE_NO),$IPO_MODE = SIPO_MODE(FP415.IPO_FRAME),$LOAD = SLOAD(FP415.TOOL_NO),$ACC = SACC_CP(LCPDAT415),$ORI_TYPE = SORI_TYP(LCPDAT415),$APO = SAPO(LCPDAT415),$JERK = SJERK(LCPDAT415),$COLLMON_TOL_PRO[1] = USE_CM_PRO_VALUES(0)
;ENDFOLD

;FOLD SLIN P416 Vel=1 m/s CPDAT416 Tool[4]:Microflown3D Base[2]:straight_sol;%{PE}
;FOLD Parameters ;%{h}
;Params IlfProvider=kukaroboter.basistech.inlineforms.movement.spline; Kuka.IsGlobalPoint=False; Kuka.PointName=P416; Kuka.BlendingEnabled=False; Kuka.MoveDataName=CPDAT416; Kuka.VelocityPath=1.000; Kuka.VelocityFieldEnabled=True; Kuka.ColDetectFieldEnabled=True; Kuka.CurrentCDSetIndex=0; Kuka.MovementParameterFieldEnabled=True; IlfCommand=SLIN
;ENDFOLD
SLIN XP416 WITH $VEL = SVEL_CP(2.0, , LCPDAT416),$TOOL = STOOL2(FP416),$BASE = SBASE(FP416.BASE_NO),$IPO_MODE = SIPO_MODE(FP416.IPO_FRAME),$LOAD = SLOAD(FP416.TOOL_NO),$ACC = SACC_CP(LCPDAT416),$ORI_TYPE = SORI_TYP(LCPDAT416),$APO = SAPO(LCPDAT416),$JERK = SJERK(LCPDAT416),$COLLMON_TOL_PRO[1] = USE_CM_PRO_VALUES(0)
;ENDFOLD

;FOLD SLIN P417 Vel=1 m/s CPDAT417 Tool[4]:Microflown3D Base[2]:straight_sol;%{PE}
;FOLD Parameters ;%{h}
;Params IlfProvider=kukaroboter.basistech.inlineforms.movement.spline; Kuka.IsGlobalPoint=False; Kuka.PointName=P417; Kuka.BlendingEnabled=False; Kuka.MoveDataName=CPDAT417; Kuka.VelocityPath=1.000; Kuka.VelocityFieldEnabled=True; Kuka.ColDetectFieldEnabled=True; Kuka.CurrentCDSetIndex=0; Kuka.MovementParameterFieldEnabled=True; IlfCommand=SLIN
;ENDFOLD
SLIN XP417 WITH $VEL = SVEL_CP(2.0, , LCPDAT417),$TOOL = STOOL2(FP417),$BASE = SBASE(FP417.BASE_NO),$IPO_MODE = SIPO_MODE(FP417.IPO_FRAME),$LOAD = SLOAD(FP417.TOOL_NO),$ACC = SACC_CP(LCPDAT417),$ORI_TYPE = SORI_TYP(LCPDAT417),$APO = SAPO(LCPDAT417),$JERK = SJERK(LCPDAT417),$COLLMON_TOL_PRO[1] = USE_CM_PRO_VALUES(0)
;ENDFOLD

;FOLD SLIN P418 Vel=1 m/s CPDAT418 Tool[4]:Microflown3D Base[2]:straight_sol;%{PE}
;FOLD Parameters ;%{h}
;Params IlfProvider=kukaroboter.basistech.inlineforms.movement.spline; Kuka.IsGlobalPoint=False; Kuka.PointName=P418; Kuka.BlendingEnabled=False; Kuka.MoveDataName=CPDAT418; Kuka.VelocityPath=1.000; Kuka.VelocityFieldEnabled=True; Kuka.ColDetectFieldEnabled=True; Kuka.CurrentCDSetIndex=0; Kuka.MovementParameterFieldEnabled=True; IlfCommand=SLIN
;ENDFOLD
SLIN XP418 WITH $VEL = SVEL_CP(2.0, , LCPDAT418),$TOOL = STOOL2(FP418),$BASE = SBASE(FP418.BASE_NO),$IPO_MODE = SIPO_MODE(FP418.IPO_FRAME),$LOAD = SLOAD(FP418.TOOL_NO),$ACC = SACC_CP(LCPDAT418),$ORI_TYPE = SORI_TYP(LCPDAT418),$APO = SAPO(LCPDAT418),$JERK = SJERK(LCPDAT418),$COLLMON_TOL_PRO[1] = USE_CM_PRO_VALUES(0)
;ENDFOLD

;FOLD SLIN P419 Vel=1 m/s CPDAT419 Tool[4]:Microflown3D Base[2]:straight_sol;%{PE}
;FOLD Parameters ;%{h}
;Params IlfProvider=kukaroboter.basistech.inlineforms.movement.spline; Kuka.IsGlobalPoint=False; Kuka.PointName=P419; Kuka.BlendingEnabled=False; Kuka.MoveDataName=CPDAT419; Kuka.VelocityPath=1.000; Kuka.VelocityFieldEnabled=True; Kuka.ColDetectFieldEnabled=True; Kuka.CurrentCDSetIndex=0; Kuka.MovementParameterFieldEnabled=True; IlfCommand=SLIN
;ENDFOLD
SLIN XP419 WITH $VEL = SVEL_CP(2.0, , LCPDAT419),$TOOL = STOOL2(FP419),$BASE = SBASE(FP419.BASE_NO),$IPO_MODE = SIPO_MODE(FP419.IPO_FRAME),$LOAD = SLOAD(FP419.TOOL_NO),$ACC = SACC_CP(LCPDAT419),$ORI_TYPE = SORI_TYP(LCPDAT419),$APO = SAPO(LCPDAT419),$JERK = SJERK(LCPDAT419),$COLLMON_TOL_PRO[1] = USE_CM_PRO_VALUES(0)
;ENDFOLD

;FOLD SLIN P420 Vel=1 m/s CPDAT420 Tool[4]:Microflown3D Base[2]:straight_sol;%{PE}
;FOLD Parameters ;%{h}
;Params IlfProvider=kukaroboter.basistech.inlineforms.movement.spline; Kuka.IsGlobalPoint=False; Kuka.PointName=P420; Kuka.BlendingEnabled=False; Kuka.MoveDataName=CPDAT420; Kuka.VelocityPath=1.000; Kuka.VelocityFieldEnabled=True; Kuka.ColDetectFieldEnabled=True; Kuka.CurrentCDSetIndex=0; Kuka.MovementParameterFieldEnabled=True; IlfCommand=SLIN
;ENDFOLD
SLIN XP420 WITH $VEL = SVEL_CP(2.0, , LCPDAT420),$TOOL = STOOL2(FP420),$BASE = SBASE(FP420.BASE_NO),$IPO_MODE = SIPO_MODE(FP420.IPO_FRAME),$LOAD = SLOAD(FP420.TOOL_NO),$ACC = SACC_CP(LCPDAT420),$ORI_TYPE = SORI_TYP(LCPDAT420),$APO = SAPO(LCPDAT420),$JERK = SJERK(LCPDAT420),$COLLMON_TOL_PRO[1] = USE_CM_PRO_VALUES(0)
;ENDFOLD

;FOLD SLIN P421 Vel=1 m/s CPDAT421 Tool[4]:Microflown3D Base[2]:straight_sol;%{PE}
;FOLD Parameters ;%{h}
;Params IlfProvider=kukaroboter.basistech.inlineforms.movement.spline; Kuka.IsGlobalPoint=False; Kuka.PointName=P421; Kuka.BlendingEnabled=False; Kuka.MoveDataName=CPDAT421; Kuka.VelocityPath=1.000; Kuka.VelocityFieldEnabled=True; Kuka.ColDetectFieldEnabled=True; Kuka.CurrentCDSetIndex=0; Kuka.MovementParameterFieldEnabled=True; IlfCommand=SLIN
;ENDFOLD
SLIN XP421 WITH $VEL = SVEL_CP(2.0, , LCPDAT421),$TOOL = STOOL2(FP421),$BASE = SBASE(FP421.BASE_NO),$IPO_MODE = SIPO_MODE(FP421.IPO_FRAME),$LOAD = SLOAD(FP421.TOOL_NO),$ACC = SACC_CP(LCPDAT421),$ORI_TYPE = SORI_TYP(LCPDAT421),$APO = SAPO(LCPDAT421),$JERK = SJERK(LCPDAT421),$COLLMON_TOL_PRO[1] = USE_CM_PRO_VALUES(0)
;ENDFOLD

;FOLD SLIN P422 Vel=1 m/s CPDAT422 Tool[4]:Microflown3D Base[2]:straight_sol;%{PE}
;FOLD Parameters ;%{h}
;Params IlfProvider=kukaroboter.basistech.inlineforms.movement.spline; Kuka.IsGlobalPoint=False; Kuka.PointName=P422; Kuka.BlendingEnabled=False; Kuka.MoveDataName=CPDAT422; Kuka.VelocityPath=1.000; Kuka.VelocityFieldEnabled=True; Kuka.ColDetectFieldEnabled=True; Kuka.CurrentCDSetIndex=0; Kuka.MovementParameterFieldEnabled=True; IlfCommand=SLIN
;ENDFOLD
SLIN XP422 WITH $VEL = SVEL_CP(2.0, , LCPDAT422),$TOOL = STOOL2(FP422),$BASE = SBASE(FP422.BASE_NO),$IPO_MODE = SIPO_MODE(FP422.IPO_FRAME),$LOAD = SLOAD(FP422.TOOL_NO),$ACC = SACC_CP(LCPDAT422),$ORI_TYPE = SORI_TYP(LCPDAT422),$APO = SAPO(LCPDAT422),$JERK = SJERK(LCPDAT422),$COLLMON_TOL_PRO[1] = USE_CM_PRO_VALUES(0)
;ENDFOLD

;FOLD SLIN P423 Vel=1 m/s CPDAT423 Tool[4]:Microflown3D Base[2]:straight_sol;%{PE}
;FOLD Parameters ;%{h}
;Params IlfProvider=kukaroboter.basistech.inlineforms.movement.spline; Kuka.IsGlobalPoint=False; Kuka.PointName=P423; Kuka.BlendingEnabled=False; Kuka.MoveDataName=CPDAT423; Kuka.VelocityPath=1.000; Kuka.VelocityFieldEnabled=True; Kuka.ColDetectFieldEnabled=True; Kuka.CurrentCDSetIndex=0; Kuka.MovementParameterFieldEnabled=True; IlfCommand=SLIN
;ENDFOLD
SLIN XP423 WITH $VEL = SVEL_CP(2.0, , LCPDAT423),$TOOL = STOOL2(FP423),$BASE = SBASE(FP423.BASE_NO),$IPO_MODE = SIPO_MODE(FP423.IPO_FRAME),$LOAD = SLOAD(FP423.TOOL_NO),$ACC = SACC_CP(LCPDAT423),$ORI_TYPE = SORI_TYP(LCPDAT423),$APO = SAPO(LCPDAT423),$JERK = SJERK(LCPDAT423),$COLLMON_TOL_PRO[1] = USE_CM_PRO_VALUES(0)
;ENDFOLD

;FOLD SLIN P424 Vel=1 m/s CPDAT424 Tool[4]:Microflown3D Base[2]:straight_sol;%{PE}
;FOLD Parameters ;%{h}
;Params IlfProvider=kukaroboter.basistech.inlineforms.movement.spline; Kuka.IsGlobalPoint=False; Kuka.PointName=P424; Kuka.BlendingEnabled=False; Kuka.MoveDataName=CPDAT424; Kuka.VelocityPath=1.000; Kuka.VelocityFieldEnabled=True; Kuka.ColDetectFieldEnabled=True; Kuka.CurrentCDSetIndex=0; Kuka.MovementParameterFieldEnabled=True; IlfCommand=SLIN
;ENDFOLD
SLIN XP424 WITH $VEL = SVEL_CP(2.0, , LCPDAT424),$TOOL = STOOL2(FP424),$BASE = SBASE(FP424.BASE_NO),$IPO_MODE = SIPO_MODE(FP424.IPO_FRAME),$LOAD = SLOAD(FP424.TOOL_NO),$ACC = SACC_CP(LCPDAT424),$ORI_TYPE = SORI_TYP(LCPDAT424),$APO = SAPO(LCPDAT424),$JERK = SJERK(LCPDAT424),$COLLMON_TOL_PRO[1] = USE_CM_PRO_VALUES(0)
;ENDFOLD

;FOLD SLIN P425 Vel=1 m/s CPDAT425 Tool[4]:Microflown3D Base[2]:straight_sol;%{PE}
;FOLD Parameters ;%{h}
;Params IlfProvider=kukaroboter.basistech.inlineforms.movement.spline; Kuka.IsGlobalPoint=False; Kuka.PointName=P425; Kuka.BlendingEnabled=False; Kuka.MoveDataName=CPDAT425; Kuka.VelocityPath=1.000; Kuka.VelocityFieldEnabled=True; Kuka.ColDetectFieldEnabled=True; Kuka.CurrentCDSetIndex=0; Kuka.MovementParameterFieldEnabled=True; IlfCommand=SLIN
;ENDFOLD
SLIN XP425 WITH $VEL = SVEL_CP(2.0, , LCPDAT425),$TOOL = STOOL2(FP425),$BASE = SBASE(FP425.BASE_NO),$IPO_MODE = SIPO_MODE(FP425.IPO_FRAME),$LOAD = SLOAD(FP425.TOOL_NO),$ACC = SACC_CP(LCPDAT425),$ORI_TYPE = SORI_TYP(LCPDAT425),$APO = SAPO(LCPDAT425),$JERK = SJERK(LCPDAT425),$COLLMON_TOL_PRO[1] = USE_CM_PRO_VALUES(0)
;ENDFOLD

;FOLD SLIN P426 Vel=1 m/s CPDAT426 Tool[4]:Microflown3D Base[2]:straight_sol;%{PE}
;FOLD Parameters ;%{h}
;Params IlfProvider=kukaroboter.basistech.inlineforms.movement.spline; Kuka.IsGlobalPoint=False; Kuka.PointName=P426; Kuka.BlendingEnabled=False; Kuka.MoveDataName=CPDAT426; Kuka.VelocityPath=1.000; Kuka.VelocityFieldEnabled=True; Kuka.ColDetectFieldEnabled=True; Kuka.CurrentCDSetIndex=0; Kuka.MovementParameterFieldEnabled=True; IlfCommand=SLIN
;ENDFOLD
SLIN XP426 WITH $VEL = SVEL_CP(2.0, , LCPDAT426),$TOOL = STOOL2(FP426),$BASE = SBASE(FP426.BASE_NO),$IPO_MODE = SIPO_MODE(FP426.IPO_FRAME),$LOAD = SLOAD(FP426.TOOL_NO),$ACC = SACC_CP(LCPDAT426),$ORI_TYPE = SORI_TYP(LCPDAT426),$APO = SAPO(LCPDAT426),$JERK = SJERK(LCPDAT426),$COLLMON_TOL_PRO[1] = USE_CM_PRO_VALUES(0)
;ENDFOLD

;FOLD SLIN P427 Vel=1 m/s CPDAT427 Tool[4]:Microflown3D Base[2]:straight_sol;%{PE}
;FOLD Parameters ;%{h}
;Params IlfProvider=kukaroboter.basistech.inlineforms.movement.spline; Kuka.IsGlobalPoint=False; Kuka.PointName=P427; Kuka.BlendingEnabled=False; Kuka.MoveDataName=CPDAT427; Kuka.VelocityPath=1.000; Kuka.VelocityFieldEnabled=True; Kuka.ColDetectFieldEnabled=True; Kuka.CurrentCDSetIndex=0; Kuka.MovementParameterFieldEnabled=True; IlfCommand=SLIN
;ENDFOLD
SLIN XP427 WITH $VEL = SVEL_CP(2.0, , LCPDAT427),$TOOL = STOOL2(FP427),$BASE = SBASE(FP427.BASE_NO),$IPO_MODE = SIPO_MODE(FP427.IPO_FRAME),$LOAD = SLOAD(FP427.TOOL_NO),$ACC = SACC_CP(LCPDAT427),$ORI_TYPE = SORI_TYP(LCPDAT427),$APO = SAPO(LCPDAT427),$JERK = SJERK(LCPDAT427),$COLLMON_TOL_PRO[1] = USE_CM_PRO_VALUES(0)
;ENDFOLD

;FOLD SLIN P428 Vel=1 m/s CPDAT428 Tool[4]:Microflown3D Base[2]:straight_sol;%{PE}
;FOLD Parameters ;%{h}
;Params IlfProvider=kukaroboter.basistech.inlineforms.movement.spline; Kuka.IsGlobalPoint=False; Kuka.PointName=P428; Kuka.BlendingEnabled=False; Kuka.MoveDataName=CPDAT428; Kuka.VelocityPath=1.000; Kuka.VelocityFieldEnabled=True; Kuka.ColDetectFieldEnabled=True; Kuka.CurrentCDSetIndex=0; Kuka.MovementParameterFieldEnabled=True; IlfCommand=SLIN
;ENDFOLD
SLIN XP428 WITH $VEL = SVEL_CP(2.0, , LCPDAT428),$TOOL = STOOL2(FP428),$BASE = SBASE(FP428.BASE_NO),$IPO_MODE = SIPO_MODE(FP428.IPO_FRAME),$LOAD = SLOAD(FP428.TOOL_NO),$ACC = SACC_CP(LCPDAT428),$ORI_TYPE = SORI_TYP(LCPDAT428),$APO = SAPO(LCPDAT428),$JERK = SJERK(LCPDAT428),$COLLMON_TOL_PRO[1] = USE_CM_PRO_VALUES(0)
;ENDFOLD

;FOLD SLIN P429 Vel=1 m/s CPDAT429 Tool[4]:Microflown3D Base[2]:straight_sol;%{PE}
;FOLD Parameters ;%{h}
;Params IlfProvider=kukaroboter.basistech.inlineforms.movement.spline; Kuka.IsGlobalPoint=False; Kuka.PointName=P429; Kuka.BlendingEnabled=False; Kuka.MoveDataName=CPDAT429; Kuka.VelocityPath=1.000; Kuka.VelocityFieldEnabled=True; Kuka.ColDetectFieldEnabled=True; Kuka.CurrentCDSetIndex=0; Kuka.MovementParameterFieldEnabled=True; IlfCommand=SLIN
;ENDFOLD
SLIN XP429 WITH $VEL = SVEL_CP(2.0, , LCPDAT429),$TOOL = STOOL2(FP429),$BASE = SBASE(FP429.BASE_NO),$IPO_MODE = SIPO_MODE(FP429.IPO_FRAME),$LOAD = SLOAD(FP429.TOOL_NO),$ACC = SACC_CP(LCPDAT429),$ORI_TYPE = SORI_TYP(LCPDAT429),$APO = SAPO(LCPDAT429),$JERK = SJERK(LCPDAT429),$COLLMON_TOL_PRO[1] = USE_CM_PRO_VALUES(0)
;ENDFOLD

;FOLD SLIN P430 Vel=1 m/s CPDAT430 Tool[4]:Microflown3D Base[2]:straight_sol;%{PE}
;FOLD Parameters ;%{h}
;Params IlfProvider=kukaroboter.basistech.inlineforms.movement.spline; Kuka.IsGlobalPoint=False; Kuka.PointName=P430; Kuka.BlendingEnabled=False; Kuka.MoveDataName=CPDAT430; Kuka.VelocityPath=1.000; Kuka.VelocityFieldEnabled=True; Kuka.ColDetectFieldEnabled=True; Kuka.CurrentCDSetIndex=0; Kuka.MovementParameterFieldEnabled=True; IlfCommand=SLIN
;ENDFOLD
SLIN XP430 WITH $VEL = SVEL_CP(2.0, , LCPDAT430),$TOOL = STOOL2(FP430),$BASE = SBASE(FP430.BASE_NO),$IPO_MODE = SIPO_MODE(FP430.IPO_FRAME),$LOAD = SLOAD(FP430.TOOL_NO),$ACC = SACC_CP(LCPDAT430),$ORI_TYPE = SORI_TYP(LCPDAT430),$APO = SAPO(LCPDAT430),$JERK = SJERK(LCPDAT430),$COLLMON_TOL_PRO[1] = USE_CM_PRO_VALUES(0)
;ENDFOLD

;FOLD SLIN P431 Vel=1 m/s CPDAT431 Tool[4]:Microflown3D Base[2]:straight_sol;%{PE}
;FOLD Parameters ;%{h}
;Params IlfProvider=kukaroboter.basistech.inlineforms.movement.spline; Kuka.IsGlobalPoint=False; Kuka.PointName=P431; Kuka.BlendingEnabled=False; Kuka.MoveDataName=CPDAT431; Kuka.VelocityPath=1.000; Kuka.VelocityFieldEnabled=True; Kuka.ColDetectFieldEnabled=True; Kuka.CurrentCDSetIndex=0; Kuka.MovementParameterFieldEnabled=True; IlfCommand=SLIN
;ENDFOLD
SLIN XP431 WITH $VEL = SVEL_CP(2.0, , LCPDAT431),$TOOL = STOOL2(FP431),$BASE = SBASE(FP431.BASE_NO),$IPO_MODE = SIPO_MODE(FP431.IPO_FRAME),$LOAD = SLOAD(FP431.TOOL_NO),$ACC = SACC_CP(LCPDAT431),$ORI_TYPE = SORI_TYP(LCPDAT431),$APO = SAPO(LCPDAT431),$JERK = SJERK(LCPDAT431),$COLLMON_TOL_PRO[1] = USE_CM_PRO_VALUES(0)
;ENDFOLD

;FOLD SLIN P432 Vel=1 m/s CPDAT432 Tool[4]:Microflown3D Base[2]:straight_sol;%{PE}
;FOLD Parameters ;%{h}
;Params IlfProvider=kukaroboter.basistech.inlineforms.movement.spline; Kuka.IsGlobalPoint=False; Kuka.PointName=P432; Kuka.BlendingEnabled=False; Kuka.MoveDataName=CPDAT432; Kuka.VelocityPath=1.000; Kuka.VelocityFieldEnabled=True; Kuka.ColDetectFieldEnabled=True; Kuka.CurrentCDSetIndex=0; Kuka.MovementParameterFieldEnabled=True; IlfCommand=SLIN
;ENDFOLD
SLIN XP432 WITH $VEL = SVEL_CP(2.0, , LCPDAT432),$TOOL = STOOL2(FP432),$BASE = SBASE(FP432.BASE_NO),$IPO_MODE = SIPO_MODE(FP432.IPO_FRAME),$LOAD = SLOAD(FP432.TOOL_NO),$ACC = SACC_CP(LCPDAT432),$ORI_TYPE = SORI_TYP(LCPDAT432),$APO = SAPO(LCPDAT432),$JERK = SJERK(LCPDAT432),$COLLMON_TOL_PRO[1] = USE_CM_PRO_VALUES(0)
;ENDFOLD

;FOLD SLIN P433 Vel=1 m/s CPDAT433 Tool[4]:Microflown3D Base[2]:straight_sol;%{PE}
;FOLD Parameters ;%{h}
;Params IlfProvider=kukaroboter.basistech.inlineforms.movement.spline; Kuka.IsGlobalPoint=False; Kuka.PointName=P433; Kuka.BlendingEnabled=False; Kuka.MoveDataName=CPDAT433; Kuka.VelocityPath=1.000; Kuka.VelocityFieldEnabled=True; Kuka.ColDetectFieldEnabled=True; Kuka.CurrentCDSetIndex=0; Kuka.MovementParameterFieldEnabled=True; IlfCommand=SLIN
;ENDFOLD
SLIN XP433 WITH $VEL = SVEL_CP(2.0, , LCPDAT433),$TOOL = STOOL2(FP433),$BASE = SBASE(FP433.BASE_NO),$IPO_MODE = SIPO_MODE(FP433.IPO_FRAME),$LOAD = SLOAD(FP433.TOOL_NO),$ACC = SACC_CP(LCPDAT433),$ORI_TYPE = SORI_TYP(LCPDAT433),$APO = SAPO(LCPDAT433),$JERK = SJERK(LCPDAT433),$COLLMON_TOL_PRO[1] = USE_CM_PRO_VALUES(0)
;ENDFOLD

;FOLD SLIN P434 Vel=1 m/s CPDAT434 Tool[4]:Microflown3D Base[2]:straight_sol;%{PE}
;FOLD Parameters ;%{h}
;Params IlfProvider=kukaroboter.basistech.inlineforms.movement.spline; Kuka.IsGlobalPoint=False; Kuka.PointName=P434; Kuka.BlendingEnabled=False; Kuka.MoveDataName=CPDAT434; Kuka.VelocityPath=1.000; Kuka.VelocityFieldEnabled=True; Kuka.ColDetectFieldEnabled=True; Kuka.CurrentCDSetIndex=0; Kuka.MovementParameterFieldEnabled=True; IlfCommand=SLIN
;ENDFOLD
SLIN XP434 WITH $VEL = SVEL_CP(2.0, , LCPDAT434),$TOOL = STOOL2(FP434),$BASE = SBASE(FP434.BASE_NO),$IPO_MODE = SIPO_MODE(FP434.IPO_FRAME),$LOAD = SLOAD(FP434.TOOL_NO),$ACC = SACC_CP(LCPDAT434),$ORI_TYPE = SORI_TYP(LCPDAT434),$APO = SAPO(LCPDAT434),$JERK = SJERK(LCPDAT434),$COLLMON_TOL_PRO[1] = USE_CM_PRO_VALUES(0)
;ENDFOLD

;FOLD SLIN P435 Vel=1 m/s CPDAT435 Tool[4]:Microflown3D Base[2]:straight_sol;%{PE}
;FOLD Parameters ;%{h}
;Params IlfProvider=kukaroboter.basistech.inlineforms.movement.spline; Kuka.IsGlobalPoint=False; Kuka.PointName=P435; Kuka.BlendingEnabled=False; Kuka.MoveDataName=CPDAT435; Kuka.VelocityPath=1.000; Kuka.VelocityFieldEnabled=True; Kuka.ColDetectFieldEnabled=True; Kuka.CurrentCDSetIndex=0; Kuka.MovementParameterFieldEnabled=True; IlfCommand=SLIN
;ENDFOLD
SLIN XP435 WITH $VEL = SVEL_CP(2.0, , LCPDAT435),$TOOL = STOOL2(FP435),$BASE = SBASE(FP435.BASE_NO),$IPO_MODE = SIPO_MODE(FP435.IPO_FRAME),$LOAD = SLOAD(FP435.TOOL_NO),$ACC = SACC_CP(LCPDAT435),$ORI_TYPE = SORI_TYP(LCPDAT435),$APO = SAPO(LCPDAT435),$JERK = SJERK(LCPDAT435),$COLLMON_TOL_PRO[1] = USE_CM_PRO_VALUES(0)
;ENDFOLD

;FOLD SLIN P436 Vel=1 m/s CPDAT436 Tool[4]:Microflown3D Base[2]:straight_sol;%{PE}
;FOLD Parameters ;%{h}
;Params IlfProvider=kukaroboter.basistech.inlineforms.movement.spline; Kuka.IsGlobalPoint=False; Kuka.PointName=P436; Kuka.BlendingEnabled=False; Kuka.MoveDataName=CPDAT436; Kuka.VelocityPath=1.000; Kuka.VelocityFieldEnabled=True; Kuka.ColDetectFieldEnabled=True; Kuka.CurrentCDSetIndex=0; Kuka.MovementParameterFieldEnabled=True; IlfCommand=SLIN
;ENDFOLD
SLIN XP436 WITH $VEL = SVEL_CP(2.0, , LCPDAT436),$TOOL = STOOL2(FP436),$BASE = SBASE(FP436.BASE_NO),$IPO_MODE = SIPO_MODE(FP436.IPO_FRAME),$LOAD = SLOAD(FP436.TOOL_NO),$ACC = SACC_CP(LCPDAT436),$ORI_TYPE = SORI_TYP(LCPDAT436),$APO = SAPO(LCPDAT436),$JERK = SJERK(LCPDAT436),$COLLMON_TOL_PRO[1] = USE_CM_PRO_VALUES(0)
;ENDFOLD

;FOLD SLIN P437 Vel=1 m/s CPDAT437 Tool[4]:Microflown3D Base[2]:straight_sol;%{PE}
;FOLD Parameters ;%{h}
;Params IlfProvider=kukaroboter.basistech.inlineforms.movement.spline; Kuka.IsGlobalPoint=False; Kuka.PointName=P437; Kuka.BlendingEnabled=False; Kuka.MoveDataName=CPDAT437; Kuka.VelocityPath=1.000; Kuka.VelocityFieldEnabled=True; Kuka.ColDetectFieldEnabled=True; Kuka.CurrentCDSetIndex=0; Kuka.MovementParameterFieldEnabled=True; IlfCommand=SLIN
;ENDFOLD
SLIN XP437 WITH $VEL = SVEL_CP(2.0, , LCPDAT437),$TOOL = STOOL2(FP437),$BASE = SBASE(FP437.BASE_NO),$IPO_MODE = SIPO_MODE(FP437.IPO_FRAME),$LOAD = SLOAD(FP437.TOOL_NO),$ACC = SACC_CP(LCPDAT437),$ORI_TYPE = SORI_TYP(LCPDAT437),$APO = SAPO(LCPDAT437),$JERK = SJERK(LCPDAT437),$COLLMON_TOL_PRO[1] = USE_CM_PRO_VALUES(0)
;ENDFOLD

;FOLD SLIN P438 Vel=1 m/s CPDAT438 Tool[4]:Microflown3D Base[2]:straight_sol;%{PE}
;FOLD Parameters ;%{h}
;Params IlfProvider=kukaroboter.basistech.inlineforms.movement.spline; Kuka.IsGlobalPoint=False; Kuka.PointName=P438; Kuka.BlendingEnabled=False; Kuka.MoveDataName=CPDAT438; Kuka.VelocityPath=1.000; Kuka.VelocityFieldEnabled=True; Kuka.ColDetectFieldEnabled=True; Kuka.CurrentCDSetIndex=0; Kuka.MovementParameterFieldEnabled=True; IlfCommand=SLIN
;ENDFOLD
SLIN XP438 WITH $VEL = SVEL_CP(2.0, , LCPDAT438),$TOOL = STOOL2(FP438),$BASE = SBASE(FP438.BASE_NO),$IPO_MODE = SIPO_MODE(FP438.IPO_FRAME),$LOAD = SLOAD(FP438.TOOL_NO),$ACC = SACC_CP(LCPDAT438),$ORI_TYPE = SORI_TYP(LCPDAT438),$APO = SAPO(LCPDAT438),$JERK = SJERK(LCPDAT438),$COLLMON_TOL_PRO[1] = USE_CM_PRO_VALUES(0)
;ENDFOLD

;FOLD SLIN P439 Vel=1 m/s CPDAT439 Tool[4]:Microflown3D Base[2]:straight_sol;%{PE}
;FOLD Parameters ;%{h}
;Params IlfProvider=kukaroboter.basistech.inlineforms.movement.spline; Kuka.IsGlobalPoint=False; Kuka.PointName=P439; Kuka.BlendingEnabled=False; Kuka.MoveDataName=CPDAT439; Kuka.VelocityPath=1.000; Kuka.VelocityFieldEnabled=True; Kuka.ColDetectFieldEnabled=True; Kuka.CurrentCDSetIndex=0; Kuka.MovementParameterFieldEnabled=True; IlfCommand=SLIN
;ENDFOLD
SLIN XP439 WITH $VEL = SVEL_CP(2.0, , LCPDAT439),$TOOL = STOOL2(FP439),$BASE = SBASE(FP439.BASE_NO),$IPO_MODE = SIPO_MODE(FP439.IPO_FRAME),$LOAD = SLOAD(FP439.TOOL_NO),$ACC = SACC_CP(LCPDAT439),$ORI_TYPE = SORI_TYP(LCPDAT439),$APO = SAPO(LCPDAT439),$JERK = SJERK(LCPDAT439),$COLLMON_TOL_PRO[1] = USE_CM_PRO_VALUES(0)
;ENDFOLD

;FOLD SLIN P440 Vel=1 m/s CPDAT440 Tool[4]:Microflown3D Base[2]:straight_sol;%{PE}
;FOLD Parameters ;%{h}
;Params IlfProvider=kukaroboter.basistech.inlineforms.movement.spline; Kuka.IsGlobalPoint=False; Kuka.PointName=P440; Kuka.BlendingEnabled=False; Kuka.MoveDataName=CPDAT440; Kuka.VelocityPath=1.000; Kuka.VelocityFieldEnabled=True; Kuka.ColDetectFieldEnabled=True; Kuka.CurrentCDSetIndex=0; Kuka.MovementParameterFieldEnabled=True; IlfCommand=SLIN
;ENDFOLD
SLIN XP440 WITH $VEL = SVEL_CP(2.0, , LCPDAT440),$TOOL = STOOL2(FP440),$BASE = SBASE(FP440.BASE_NO),$IPO_MODE = SIPO_MODE(FP440.IPO_FRAME),$LOAD = SLOAD(FP440.TOOL_NO),$ACC = SACC_CP(LCPDAT440),$ORI_TYPE = SORI_TYP(LCPDAT440),$APO = SAPO(LCPDAT440),$JERK = SJERK(LCPDAT440),$COLLMON_TOL_PRO[1] = USE_CM_PRO_VALUES(0)
;ENDFOLD

;FOLD SLIN P441 Vel=1 m/s CPDAT441 Tool[4]:Microflown3D Base[2]:straight_sol;%{PE}
;FOLD Parameters ;%{h}
;Params IlfProvider=kukaroboter.basistech.inlineforms.movement.spline; Kuka.IsGlobalPoint=False; Kuka.PointName=P441; Kuka.BlendingEnabled=False; Kuka.MoveDataName=CPDAT441; Kuka.VelocityPath=1.000; Kuka.VelocityFieldEnabled=True; Kuka.ColDetectFieldEnabled=True; Kuka.CurrentCDSetIndex=0; Kuka.MovementParameterFieldEnabled=True; IlfCommand=SLIN
;ENDFOLD
SLIN XP441 WITH $VEL = SVEL_CP(2.0, , LCPDAT441),$TOOL = STOOL2(FP441),$BASE = SBASE(FP441.BASE_NO),$IPO_MODE = SIPO_MODE(FP441.IPO_FRAME),$LOAD = SLOAD(FP441.TOOL_NO),$ACC = SACC_CP(LCPDAT441),$ORI_TYPE = SORI_TYP(LCPDAT441),$APO = SAPO(LCPDAT441),$JERK = SJERK(LCPDAT441),$COLLMON_TOL_PRO[1] = USE_CM_PRO_VALUES(0)
;ENDFOLD

;FOLD SLIN P442 Vel=1 m/s CPDAT442 Tool[4]:Microflown3D Base[2]:straight_sol;%{PE}
;FOLD Parameters ;%{h}
;Params IlfProvider=kukaroboter.basistech.inlineforms.movement.spline; Kuka.IsGlobalPoint=False; Kuka.PointName=P442; Kuka.BlendingEnabled=False; Kuka.MoveDataName=CPDAT442; Kuka.VelocityPath=1.000; Kuka.VelocityFieldEnabled=True; Kuka.ColDetectFieldEnabled=True; Kuka.CurrentCDSetIndex=0; Kuka.MovementParameterFieldEnabled=True; IlfCommand=SLIN
;ENDFOLD
SLIN XP442 WITH $VEL = SVEL_CP(2.0, , LCPDAT442),$TOOL = STOOL2(FP442),$BASE = SBASE(FP442.BASE_NO),$IPO_MODE = SIPO_MODE(FP442.IPO_FRAME),$LOAD = SLOAD(FP442.TOOL_NO),$ACC = SACC_CP(LCPDAT442),$ORI_TYPE = SORI_TYP(LCPDAT442),$APO = SAPO(LCPDAT442),$JERK = SJERK(LCPDAT442),$COLLMON_TOL_PRO[1] = USE_CM_PRO_VALUES(0)
;ENDFOLD

;FOLD SLIN P443 Vel=1 m/s CPDAT443 Tool[4]:Microflown3D Base[2]:straight_sol;%{PE}
;FOLD Parameters ;%{h}
;Params IlfProvider=kukaroboter.basistech.inlineforms.movement.spline; Kuka.IsGlobalPoint=False; Kuka.PointName=P443; Kuka.BlendingEnabled=False; Kuka.MoveDataName=CPDAT443; Kuka.VelocityPath=1.000; Kuka.VelocityFieldEnabled=True; Kuka.ColDetectFieldEnabled=True; Kuka.CurrentCDSetIndex=0; Kuka.MovementParameterFieldEnabled=True; IlfCommand=SLIN
;ENDFOLD
SLIN XP443 WITH $VEL = SVEL_CP(2.0, , LCPDAT443),$TOOL = STOOL2(FP443),$BASE = SBASE(FP443.BASE_NO),$IPO_MODE = SIPO_MODE(FP443.IPO_FRAME),$LOAD = SLOAD(FP443.TOOL_NO),$ACC = SACC_CP(LCPDAT443),$ORI_TYPE = SORI_TYP(LCPDAT443),$APO = SAPO(LCPDAT443),$JERK = SJERK(LCPDAT443),$COLLMON_TOL_PRO[1] = USE_CM_PRO_VALUES(0)
;ENDFOLD

;FOLD SLIN P444 Vel=1 m/s CPDAT444 Tool[4]:Microflown3D Base[2]:straight_sol;%{PE}
;FOLD Parameters ;%{h}
;Params IlfProvider=kukaroboter.basistech.inlineforms.movement.spline; Kuka.IsGlobalPoint=False; Kuka.PointName=P444; Kuka.BlendingEnabled=False; Kuka.MoveDataName=CPDAT444; Kuka.VelocityPath=1.000; Kuka.VelocityFieldEnabled=True; Kuka.ColDetectFieldEnabled=True; Kuka.CurrentCDSetIndex=0; Kuka.MovementParameterFieldEnabled=True; IlfCommand=SLIN
;ENDFOLD
SLIN XP444 WITH $VEL = SVEL_CP(2.0, , LCPDAT444),$TOOL = STOOL2(FP444),$BASE = SBASE(FP444.BASE_NO),$IPO_MODE = SIPO_MODE(FP444.IPO_FRAME),$LOAD = SLOAD(FP444.TOOL_NO),$ACC = SACC_CP(LCPDAT444),$ORI_TYPE = SORI_TYP(LCPDAT444),$APO = SAPO(LCPDAT444),$JERK = SJERK(LCPDAT444),$COLLMON_TOL_PRO[1] = USE_CM_PRO_VALUES(0)
;ENDFOLD

;FOLD SLIN P445 Vel=1 m/s CPDAT445 Tool[4]:Microflown3D Base[2]:straight_sol;%{PE}
;FOLD Parameters ;%{h}
;Params IlfProvider=kukaroboter.basistech.inlineforms.movement.spline; Kuka.IsGlobalPoint=False; Kuka.PointName=P445; Kuka.BlendingEnabled=False; Kuka.MoveDataName=CPDAT445; Kuka.VelocityPath=1.000; Kuka.VelocityFieldEnabled=True; Kuka.ColDetectFieldEnabled=True; Kuka.CurrentCDSetIndex=0; Kuka.MovementParameterFieldEnabled=True; IlfCommand=SLIN
;ENDFOLD
SLIN XP445 WITH $VEL = SVEL_CP(2.0, , LCPDAT445),$TOOL = STOOL2(FP445),$BASE = SBASE(FP445.BASE_NO),$IPO_MODE = SIPO_MODE(FP445.IPO_FRAME),$LOAD = SLOAD(FP445.TOOL_NO),$ACC = SACC_CP(LCPDAT445),$ORI_TYPE = SORI_TYP(LCPDAT445),$APO = SAPO(LCPDAT445),$JERK = SJERK(LCPDAT445),$COLLMON_TOL_PRO[1] = USE_CM_PRO_VALUES(0)
;ENDFOLD

;FOLD SLIN P446 Vel=1 m/s CPDAT446 Tool[4]:Microflown3D Base[2]:straight_sol;%{PE}
;FOLD Parameters ;%{h}
;Params IlfProvider=kukaroboter.basistech.inlineforms.movement.spline; Kuka.IsGlobalPoint=False; Kuka.PointName=P446; Kuka.BlendingEnabled=False; Kuka.MoveDataName=CPDAT446; Kuka.VelocityPath=1.000; Kuka.VelocityFieldEnabled=True; Kuka.ColDetectFieldEnabled=True; Kuka.CurrentCDSetIndex=0; Kuka.MovementParameterFieldEnabled=True; IlfCommand=SLIN
;ENDFOLD
SLIN XP446 WITH $VEL = SVEL_CP(2.0, , LCPDAT446),$TOOL = STOOL2(FP446),$BASE = SBASE(FP446.BASE_NO),$IPO_MODE = SIPO_MODE(FP446.IPO_FRAME),$LOAD = SLOAD(FP446.TOOL_NO),$ACC = SACC_CP(LCPDAT446),$ORI_TYPE = SORI_TYP(LCPDAT446),$APO = SAPO(LCPDAT446),$JERK = SJERK(LCPDAT446),$COLLMON_TOL_PRO[1] = USE_CM_PRO_VALUES(0)
;ENDFOLD

;FOLD SLIN P447 Vel=1 m/s CPDAT447 Tool[4]:Microflown3D Base[2]:straight_sol;%{PE}
;FOLD Parameters ;%{h}
;Params IlfProvider=kukaroboter.basistech.inlineforms.movement.spline; Kuka.IsGlobalPoint=False; Kuka.PointName=P447; Kuka.BlendingEnabled=False; Kuka.MoveDataName=CPDAT447; Kuka.VelocityPath=1.000; Kuka.VelocityFieldEnabled=True; Kuka.ColDetectFieldEnabled=True; Kuka.CurrentCDSetIndex=0; Kuka.MovementParameterFieldEnabled=True; IlfCommand=SLIN
;ENDFOLD
SLIN XP447 WITH $VEL = SVEL_CP(2.0, , LCPDAT447),$TOOL = STOOL2(FP447),$BASE = SBASE(FP447.BASE_NO),$IPO_MODE = SIPO_MODE(FP447.IPO_FRAME),$LOAD = SLOAD(FP447.TOOL_NO),$ACC = SACC_CP(LCPDAT447),$ORI_TYPE = SORI_TYP(LCPDAT447),$APO = SAPO(LCPDAT447),$JERK = SJERK(LCPDAT447),$COLLMON_TOL_PRO[1] = USE_CM_PRO_VALUES(0)
;ENDFOLD

;FOLD SLIN P448 Vel=1 m/s CPDAT448 Tool[4]:Microflown3D Base[2]:straight_sol;%{PE}
;FOLD Parameters ;%{h}
;Params IlfProvider=kukaroboter.basistech.inlineforms.movement.spline; Kuka.IsGlobalPoint=False; Kuka.PointName=P448; Kuka.BlendingEnabled=False; Kuka.MoveDataName=CPDAT448; Kuka.VelocityPath=1.000; Kuka.VelocityFieldEnabled=True; Kuka.ColDetectFieldEnabled=True; Kuka.CurrentCDSetIndex=0; Kuka.MovementParameterFieldEnabled=True; IlfCommand=SLIN
;ENDFOLD
SLIN XP448 WITH $VEL = SVEL_CP(2.0, , LCPDAT448),$TOOL = STOOL2(FP448),$BASE = SBASE(FP448.BASE_NO),$IPO_MODE = SIPO_MODE(FP448.IPO_FRAME),$LOAD = SLOAD(FP448.TOOL_NO),$ACC = SACC_CP(LCPDAT448),$ORI_TYPE = SORI_TYP(LCPDAT448),$APO = SAPO(LCPDAT448),$JERK = SJERK(LCPDAT448),$COLLMON_TOL_PRO[1] = USE_CM_PRO_VALUES(0)
;ENDFOLD

;FOLD SLIN P449 Vel=1 m/s CPDAT449 Tool[4]:Microflown3D Base[2]:straight_sol;%{PE}
;FOLD Parameters ;%{h}
;Params IlfProvider=kukaroboter.basistech.inlineforms.movement.spline; Kuka.IsGlobalPoint=False; Kuka.PointName=P449; Kuka.BlendingEnabled=False; Kuka.MoveDataName=CPDAT449; Kuka.VelocityPath=1.000; Kuka.VelocityFieldEnabled=True; Kuka.ColDetectFieldEnabled=True; Kuka.CurrentCDSetIndex=0; Kuka.MovementParameterFieldEnabled=True; IlfCommand=SLIN
;ENDFOLD
SLIN XP449 WITH $VEL = SVEL_CP(2.0, , LCPDAT449),$TOOL = STOOL2(FP449),$BASE = SBASE(FP449.BASE_NO),$IPO_MODE = SIPO_MODE(FP449.IPO_FRAME),$LOAD = SLOAD(FP449.TOOL_NO),$ACC = SACC_CP(LCPDAT449),$ORI_TYPE = SORI_TYP(LCPDAT449),$APO = SAPO(LCPDAT449),$JERK = SJERK(LCPDAT449),$COLLMON_TOL_PRO[1] = USE_CM_PRO_VALUES(0)
;ENDFOLD

;FOLD SLIN P450 Vel=1 m/s CPDAT450 Tool[4]:Microflown3D Base[2]:straight_sol;%{PE}
;FOLD Parameters ;%{h}
;Params IlfProvider=kukaroboter.basistech.inlineforms.movement.spline; Kuka.IsGlobalPoint=False; Kuka.PointName=P450; Kuka.BlendingEnabled=False; Kuka.MoveDataName=CPDAT450; Kuka.VelocityPath=1.000; Kuka.VelocityFieldEnabled=True; Kuka.ColDetectFieldEnabled=True; Kuka.CurrentCDSetIndex=0; Kuka.MovementParameterFieldEnabled=True; IlfCommand=SLIN
;ENDFOLD
SLIN XP450 WITH $VEL = SVEL_CP(2.0, , LCPDAT450),$TOOL = STOOL2(FP450),$BASE = SBASE(FP450.BASE_NO),$IPO_MODE = SIPO_MODE(FP450.IPO_FRAME),$LOAD = SLOAD(FP450.TOOL_NO),$ACC = SACC_CP(LCPDAT450),$ORI_TYPE = SORI_TYP(LCPDAT450),$APO = SAPO(LCPDAT450),$JERK = SJERK(LCPDAT450),$COLLMON_TOL_PRO[1] = USE_CM_PRO_VALUES(0)
;ENDFOLD

;FOLD SLIN P451 Vel=1 m/s CPDAT451 Tool[4]:Microflown3D Base[2]:straight_sol;%{PE}
;FOLD Parameters ;%{h}
;Params IlfProvider=kukaroboter.basistech.inlineforms.movement.spline; Kuka.IsGlobalPoint=False; Kuka.PointName=P451; Kuka.BlendingEnabled=False; Kuka.MoveDataName=CPDAT451; Kuka.VelocityPath=1.000; Kuka.VelocityFieldEnabled=True; Kuka.ColDetectFieldEnabled=True; Kuka.CurrentCDSetIndex=0; Kuka.MovementParameterFieldEnabled=True; IlfCommand=SLIN
;ENDFOLD
SLIN XP451 WITH $VEL = SVEL_CP(2.0, , LCPDAT451),$TOOL = STOOL2(FP451),$BASE = SBASE(FP451.BASE_NO),$IPO_MODE = SIPO_MODE(FP451.IPO_FRAME),$LOAD = SLOAD(FP451.TOOL_NO),$ACC = SACC_CP(LCPDAT451),$ORI_TYPE = SORI_TYP(LCPDAT451),$APO = SAPO(LCPDAT451),$JERK = SJERK(LCPDAT451),$COLLMON_TOL_PRO[1] = USE_CM_PRO_VALUES(0)
;ENDFOLD

;FOLD SLIN P452 Vel=1 m/s CPDAT452 Tool[4]:Microflown3D Base[2]:straight_sol;%{PE}
;FOLD Parameters ;%{h}
;Params IlfProvider=kukaroboter.basistech.inlineforms.movement.spline; Kuka.IsGlobalPoint=False; Kuka.PointName=P452; Kuka.BlendingEnabled=False; Kuka.MoveDataName=CPDAT452; Kuka.VelocityPath=1.000; Kuka.VelocityFieldEnabled=True; Kuka.ColDetectFieldEnabled=True; Kuka.CurrentCDSetIndex=0; Kuka.MovementParameterFieldEnabled=True; IlfCommand=SLIN
;ENDFOLD
SLIN XP452 WITH $VEL = SVEL_CP(2.0, , LCPDAT452),$TOOL = STOOL2(FP452),$BASE = SBASE(FP452.BASE_NO),$IPO_MODE = SIPO_MODE(FP452.IPO_FRAME),$LOAD = SLOAD(FP452.TOOL_NO),$ACC = SACC_CP(LCPDAT452),$ORI_TYPE = SORI_TYP(LCPDAT452),$APO = SAPO(LCPDAT452),$JERK = SJERK(LCPDAT452),$COLLMON_TOL_PRO[1] = USE_CM_PRO_VALUES(0)
;ENDFOLD

;FOLD SLIN P453 Vel=1 m/s CPDAT453 Tool[4]:Microflown3D Base[2]:straight_sol;%{PE}
;FOLD Parameters ;%{h}
;Params IlfProvider=kukaroboter.basistech.inlineforms.movement.spline; Kuka.IsGlobalPoint=False; Kuka.PointName=P453; Kuka.BlendingEnabled=False; Kuka.MoveDataName=CPDAT453; Kuka.VelocityPath=1.000; Kuka.VelocityFieldEnabled=True; Kuka.ColDetectFieldEnabled=True; Kuka.CurrentCDSetIndex=0; Kuka.MovementParameterFieldEnabled=True; IlfCommand=SLIN
;ENDFOLD
SLIN XP453 WITH $VEL = SVEL_CP(2.0, , LCPDAT453),$TOOL = STOOL2(FP453),$BASE = SBASE(FP453.BASE_NO),$IPO_MODE = SIPO_MODE(FP453.IPO_FRAME),$LOAD = SLOAD(FP453.TOOL_NO),$ACC = SACC_CP(LCPDAT453),$ORI_TYPE = SORI_TYP(LCPDAT453),$APO = SAPO(LCPDAT453),$JERK = SJERK(LCPDAT453),$COLLMON_TOL_PRO[1] = USE_CM_PRO_VALUES(0)
;ENDFOLD

;FOLD SLIN P454 Vel=1 m/s CPDAT454 Tool[4]:Microflown3D Base[2]:straight_sol;%{PE}
;FOLD Parameters ;%{h}
;Params IlfProvider=kukaroboter.basistech.inlineforms.movement.spline; Kuka.IsGlobalPoint=False; Kuka.PointName=P454; Kuka.BlendingEnabled=False; Kuka.MoveDataName=CPDAT454; Kuka.VelocityPath=1.000; Kuka.VelocityFieldEnabled=True; Kuka.ColDetectFieldEnabled=True; Kuka.CurrentCDSetIndex=0; Kuka.MovementParameterFieldEnabled=True; IlfCommand=SLIN
;ENDFOLD
SLIN XP454 WITH $VEL = SVEL_CP(2.0, , LCPDAT454),$TOOL = STOOL2(FP454),$BASE = SBASE(FP454.BASE_NO),$IPO_MODE = SIPO_MODE(FP454.IPO_FRAME),$LOAD = SLOAD(FP454.TOOL_NO),$ACC = SACC_CP(LCPDAT454),$ORI_TYPE = SORI_TYP(LCPDAT454),$APO = SAPO(LCPDAT454),$JERK = SJERK(LCPDAT454),$COLLMON_TOL_PRO[1] = USE_CM_PRO_VALUES(0)
;ENDFOLD

;FOLD SLIN P455 Vel=1 m/s CPDAT455 Tool[4]:Microflown3D Base[2]:straight_sol;%{PE}
;FOLD Parameters ;%{h}
;Params IlfProvider=kukaroboter.basistech.inlineforms.movement.spline; Kuka.IsGlobalPoint=False; Kuka.PointName=P455; Kuka.BlendingEnabled=False; Kuka.MoveDataName=CPDAT455; Kuka.VelocityPath=1.000; Kuka.VelocityFieldEnabled=True; Kuka.ColDetectFieldEnabled=True; Kuka.CurrentCDSetIndex=0; Kuka.MovementParameterFieldEnabled=True; IlfCommand=SLIN
;ENDFOLD
SLIN XP455 WITH $VEL = SVEL_CP(2.0, , LCPDAT455),$TOOL = STOOL2(FP455),$BASE = SBASE(FP455.BASE_NO),$IPO_MODE = SIPO_MODE(FP455.IPO_FRAME),$LOAD = SLOAD(FP455.TOOL_NO),$ACC = SACC_CP(LCPDAT455),$ORI_TYPE = SORI_TYP(LCPDAT455),$APO = SAPO(LCPDAT455),$JERK = SJERK(LCPDAT455),$COLLMON_TOL_PRO[1] = USE_CM_PRO_VALUES(0)
;ENDFOLD

;FOLD SLIN P456 Vel=1 m/s CPDAT456 Tool[4]:Microflown3D Base[2]:straight_sol;%{PE}
;FOLD Parameters ;%{h}
;Params IlfProvider=kukaroboter.basistech.inlineforms.movement.spline; Kuka.IsGlobalPoint=False; Kuka.PointName=P456; Kuka.BlendingEnabled=False; Kuka.MoveDataName=CPDAT456; Kuka.VelocityPath=1.000; Kuka.VelocityFieldEnabled=True; Kuka.ColDetectFieldEnabled=True; Kuka.CurrentCDSetIndex=0; Kuka.MovementParameterFieldEnabled=True; IlfCommand=SLIN
;ENDFOLD
SLIN XP456 WITH $VEL = SVEL_CP(2.0, , LCPDAT456),$TOOL = STOOL2(FP456),$BASE = SBASE(FP456.BASE_NO),$IPO_MODE = SIPO_MODE(FP456.IPO_FRAME),$LOAD = SLOAD(FP456.TOOL_NO),$ACC = SACC_CP(LCPDAT456),$ORI_TYPE = SORI_TYP(LCPDAT456),$APO = SAPO(LCPDAT456),$JERK = SJERK(LCPDAT456),$COLLMON_TOL_PRO[1] = USE_CM_PRO_VALUES(0)
;ENDFOLD

;FOLD SLIN P457 Vel=1 m/s CPDAT457 Tool[4]:Microflown3D Base[2]:straight_sol;%{PE}
;FOLD Parameters ;%{h}
;Params IlfProvider=kukaroboter.basistech.inlineforms.movement.spline; Kuka.IsGlobalPoint=False; Kuka.PointName=P457; Kuka.BlendingEnabled=False; Kuka.MoveDataName=CPDAT457; Kuka.VelocityPath=1.000; Kuka.VelocityFieldEnabled=True; Kuka.ColDetectFieldEnabled=True; Kuka.CurrentCDSetIndex=0; Kuka.MovementParameterFieldEnabled=True; IlfCommand=SLIN
;ENDFOLD
SLIN XP457 WITH $VEL = SVEL_CP(2.0, , LCPDAT457),$TOOL = STOOL2(FP457),$BASE = SBASE(FP457.BASE_NO),$IPO_MODE = SIPO_MODE(FP457.IPO_FRAME),$LOAD = SLOAD(FP457.TOOL_NO),$ACC = SACC_CP(LCPDAT457),$ORI_TYPE = SORI_TYP(LCPDAT457),$APO = SAPO(LCPDAT457),$JERK = SJERK(LCPDAT457),$COLLMON_TOL_PRO[1] = USE_CM_PRO_VALUES(0)
;ENDFOLD

;FOLD SLIN P458 Vel=1 m/s CPDAT458 Tool[4]:Microflown3D Base[2]:straight_sol;%{PE}
;FOLD Parameters ;%{h}
;Params IlfProvider=kukaroboter.basistech.inlineforms.movement.spline; Kuka.IsGlobalPoint=False; Kuka.PointName=P458; Kuka.BlendingEnabled=False; Kuka.MoveDataName=CPDAT458; Kuka.VelocityPath=1.000; Kuka.VelocityFieldEnabled=True; Kuka.ColDetectFieldEnabled=True; Kuka.CurrentCDSetIndex=0; Kuka.MovementParameterFieldEnabled=True; IlfCommand=SLIN
;ENDFOLD
SLIN XP458 WITH $VEL = SVEL_CP(2.0, , LCPDAT458),$TOOL = STOOL2(FP458),$BASE = SBASE(FP458.BASE_NO),$IPO_MODE = SIPO_MODE(FP458.IPO_FRAME),$LOAD = SLOAD(FP458.TOOL_NO),$ACC = SACC_CP(LCPDAT458),$ORI_TYPE = SORI_TYP(LCPDAT458),$APO = SAPO(LCPDAT458),$JERK = SJERK(LCPDAT458),$COLLMON_TOL_PRO[1] = USE_CM_PRO_VALUES(0)
;ENDFOLD

;FOLD SLIN P459 Vel=1 m/s CPDAT459 Tool[4]:Microflown3D Base[2]:straight_sol;%{PE}
;FOLD Parameters ;%{h}
;Params IlfProvider=kukaroboter.basistech.inlineforms.movement.spline; Kuka.IsGlobalPoint=False; Kuka.PointName=P459; Kuka.BlendingEnabled=False; Kuka.MoveDataName=CPDAT459; Kuka.VelocityPath=1.000; Kuka.VelocityFieldEnabled=True; Kuka.ColDetectFieldEnabled=True; Kuka.CurrentCDSetIndex=0; Kuka.MovementParameterFieldEnabled=True; IlfCommand=SLIN
;ENDFOLD
SLIN XP459 WITH $VEL = SVEL_CP(2.0, , LCPDAT459),$TOOL = STOOL2(FP459),$BASE = SBASE(FP459.BASE_NO),$IPO_MODE = SIPO_MODE(FP459.IPO_FRAME),$LOAD = SLOAD(FP459.TOOL_NO),$ACC = SACC_CP(LCPDAT459),$ORI_TYPE = SORI_TYP(LCPDAT459),$APO = SAPO(LCPDAT459),$JERK = SJERK(LCPDAT459),$COLLMON_TOL_PRO[1] = USE_CM_PRO_VALUES(0)
;ENDFOLD

;FOLD SLIN P460 Vel=1 m/s CPDAT460 Tool[4]:Microflown3D Base[2]:straight_sol;%{PE}
;FOLD Parameters ;%{h}
;Params IlfProvider=kukaroboter.basistech.inlineforms.movement.spline; Kuka.IsGlobalPoint=False; Kuka.PointName=P460; Kuka.BlendingEnabled=False; Kuka.MoveDataName=CPDAT460; Kuka.VelocityPath=1.000; Kuka.VelocityFieldEnabled=True; Kuka.ColDetectFieldEnabled=True; Kuka.CurrentCDSetIndex=0; Kuka.MovementParameterFieldEnabled=True; IlfCommand=SLIN
;ENDFOLD
SLIN XP460 WITH $VEL = SVEL_CP(2.0, , LCPDAT460),$TOOL = STOOL2(FP460),$BASE = SBASE(FP460.BASE_NO),$IPO_MODE = SIPO_MODE(FP460.IPO_FRAME),$LOAD = SLOAD(FP460.TOOL_NO),$ACC = SACC_CP(LCPDAT460),$ORI_TYPE = SORI_TYP(LCPDAT460),$APO = SAPO(LCPDAT460),$JERK = SJERK(LCPDAT460),$COLLMON_TOL_PRO[1] = USE_CM_PRO_VALUES(0)
;ENDFOLD

;FOLD SLIN P461 Vel=0.25 m/s CPDAT461 Tool[4]:Microflown3D Base[2]:straight_sol;%{PE}
;FOLD Parameters ;%{h}
;Params IlfProvider=kukaroboter.basistech.inlineforms.movement.spline; Kuka.IsGlobalPoint=False; Kuka.PointName=P461; Kuka.BlendingEnabled=False; Kuka.MoveDataName=CPDAT461; Kuka.VelocityPath=0.250; Kuka.VelocityFieldEnabled=True; Kuka.ColDetectFieldEnabled=True; Kuka.CurrentCDSetIndex=0; Kuka.MovementParameterFieldEnabled=True; IlfCommand=SLIN
;ENDFOLD
SLIN XP461 WITH $VEL = SVEL_CP(2.0, , LCPDAT461),$TOOL = STOOL2(FP461),$BASE = SBASE(FP461.BASE_NO),$IPO_MODE = SIPO_MODE(FP461.IPO_FRAME),$LOAD = SLOAD(FP461.TOOL_NO),$ACC = SACC_CP(LCPDAT461),$ORI_TYPE = SORI_TYP(LCPDAT461),$APO = SAPO(LCPDAT461),$JERK = SJERK(LCPDAT461),$COLLMON_TOL_PRO[1] = USE_CM_PRO_VALUES(0)
;ENDFOLD

;FOLD SLIN P462 Vel=0.25 m/s CPDAT462 Tool[4]:Microflown3D Base[2]:straight_sol;%{PE}
;FOLD Parameters ;%{h}
;Params IlfProvider=kukaroboter.basistech.inlineforms.movement.spline; Kuka.IsGlobalPoint=False; Kuka.PointName=P462; Kuka.BlendingEnabled=False; Kuka.MoveDataName=CPDAT462; Kuka.VelocityPath=0.250; Kuka.VelocityFieldEnabled=True; Kuka.ColDetectFieldEnabled=True; Kuka.CurrentCDSetIndex=0; Kuka.MovementParameterFieldEnabled=True; IlfCommand=SLIN
;ENDFOLD
SLIN XP462 WITH $VEL = SVEL_CP(2.0, , LCPDAT462),$TOOL = STOOL2(FP462),$BASE = SBASE(FP462.BASE_NO),$IPO_MODE = SIPO_MODE(FP462.IPO_FRAME),$LOAD = SLOAD(FP462.TOOL_NO),$ACC = SACC_CP(LCPDAT462),$ORI_TYPE = SORI_TYP(LCPDAT462),$APO = SAPO(LCPDAT462),$JERK = SJERK(LCPDAT462),$COLLMON_TOL_PRO[1] = USE_CM_PRO_VALUES(0)
;ENDFOLD

;FOLD SLIN P463 Vel=1 m/s CPDAT463 Tool[4]:Microflown3D Base[2]:straight_sol;%{PE}
;FOLD Parameters ;%{h}
;Params IlfProvider=kukaroboter.basistech.inlineforms.movement.spline; Kuka.IsGlobalPoint=False; Kuka.PointName=P463; Kuka.BlendingEnabled=False; Kuka.MoveDataName=CPDAT463; Kuka.VelocityPath=1.000; Kuka.VelocityFieldEnabled=True; Kuka.ColDetectFieldEnabled=True; Kuka.CurrentCDSetIndex=0; Kuka.MovementParameterFieldEnabled=True; IlfCommand=SLIN
;ENDFOLD
SLIN XP463 WITH $VEL = SVEL_CP(2.0, , LCPDAT463),$TOOL = STOOL2(FP463),$BASE = SBASE(FP463.BASE_NO),$IPO_MODE = SIPO_MODE(FP463.IPO_FRAME),$LOAD = SLOAD(FP463.TOOL_NO),$ACC = SACC_CP(LCPDAT463),$ORI_TYPE = SORI_TYP(LCPDAT463),$APO = SAPO(LCPDAT463),$JERK = SJERK(LCPDAT463),$COLLMON_TOL_PRO[1] = USE_CM_PRO_VALUES(0)
;ENDFOLD

;FOLD SLIN P464 Vel=1 m/s CPDAT464 Tool[4]:Microflown3D Base[2]:straight_sol;%{PE}
;FOLD Parameters ;%{h}
;Params IlfProvider=kukaroboter.basistech.inlineforms.movement.spline; Kuka.IsGlobalPoint=False; Kuka.PointName=P464; Kuka.BlendingEnabled=False; Kuka.MoveDataName=CPDAT464; Kuka.VelocityPath=1.000; Kuka.VelocityFieldEnabled=True; Kuka.ColDetectFieldEnabled=True; Kuka.CurrentCDSetIndex=0; Kuka.MovementParameterFieldEnabled=True; IlfCommand=SLIN
;ENDFOLD
SLIN XP464 WITH $VEL = SVEL_CP(2.0, , LCPDAT464),$TOOL = STOOL2(FP464),$BASE = SBASE(FP464.BASE_NO),$IPO_MODE = SIPO_MODE(FP464.IPO_FRAME),$LOAD = SLOAD(FP464.TOOL_NO),$ACC = SACC_CP(LCPDAT464),$ORI_TYPE = SORI_TYP(LCPDAT464),$APO = SAPO(LCPDAT464),$JERK = SJERK(LCPDAT464),$COLLMON_TOL_PRO[1] = USE_CM_PRO_VALUES(0)
;ENDFOLD

;FOLD SLIN P465 Vel=1 m/s CPDAT465 Tool[4]:Microflown3D Base[2]:straight_sol;%{PE}
;FOLD Parameters ;%{h}
;Params IlfProvider=kukaroboter.basistech.inlineforms.movement.spline; Kuka.IsGlobalPoint=False; Kuka.PointName=P465; Kuka.BlendingEnabled=False; Kuka.MoveDataName=CPDAT465; Kuka.VelocityPath=1.000; Kuka.VelocityFieldEnabled=True; Kuka.ColDetectFieldEnabled=True; Kuka.CurrentCDSetIndex=0; Kuka.MovementParameterFieldEnabled=True; IlfCommand=SLIN
;ENDFOLD
SLIN XP465 WITH $VEL = SVEL_CP(2.0, , LCPDAT465),$TOOL = STOOL2(FP465),$BASE = SBASE(FP465.BASE_NO),$IPO_MODE = SIPO_MODE(FP465.IPO_FRAME),$LOAD = SLOAD(FP465.TOOL_NO),$ACC = SACC_CP(LCPDAT465),$ORI_TYPE = SORI_TYP(LCPDAT465),$APO = SAPO(LCPDAT465),$JERK = SJERK(LCPDAT465),$COLLMON_TOL_PRO[1] = USE_CM_PRO_VALUES(0)
;ENDFOLD

;FOLD SLIN P466 Vel=1 m/s CPDAT466 Tool[4]:Microflown3D Base[2]:straight_sol;%{PE}
;FOLD Parameters ;%{h}
;Params IlfProvider=kukaroboter.basistech.inlineforms.movement.spline; Kuka.IsGlobalPoint=False; Kuka.PointName=P466; Kuka.BlendingEnabled=False; Kuka.MoveDataName=CPDAT466; Kuka.VelocityPath=1.000; Kuka.VelocityFieldEnabled=True; Kuka.ColDetectFieldEnabled=True; Kuka.CurrentCDSetIndex=0; Kuka.MovementParameterFieldEnabled=True; IlfCommand=SLIN
;ENDFOLD
SLIN XP466 WITH $VEL = SVEL_CP(2.0, , LCPDAT466),$TOOL = STOOL2(FP466),$BASE = SBASE(FP466.BASE_NO),$IPO_MODE = SIPO_MODE(FP466.IPO_FRAME),$LOAD = SLOAD(FP466.TOOL_NO),$ACC = SACC_CP(LCPDAT466),$ORI_TYPE = SORI_TYP(LCPDAT466),$APO = SAPO(LCPDAT466),$JERK = SJERK(LCPDAT466),$COLLMON_TOL_PRO[1] = USE_CM_PRO_VALUES(0)
;ENDFOLD

;FOLD SLIN P467 Vel=1 m/s CPDAT467 Tool[4]:Microflown3D Base[2]:straight_sol;%{PE}
;FOLD Parameters ;%{h}
;Params IlfProvider=kukaroboter.basistech.inlineforms.movement.spline; Kuka.IsGlobalPoint=False; Kuka.PointName=P467; Kuka.BlendingEnabled=False; Kuka.MoveDataName=CPDAT467; Kuka.VelocityPath=1.000; Kuka.VelocityFieldEnabled=True; Kuka.ColDetectFieldEnabled=True; Kuka.CurrentCDSetIndex=0; Kuka.MovementParameterFieldEnabled=True; IlfCommand=SLIN
;ENDFOLD
SLIN XP467 WITH $VEL = SVEL_CP(2.0, , LCPDAT467),$TOOL = STOOL2(FP467),$BASE = SBASE(FP467.BASE_NO),$IPO_MODE = SIPO_MODE(FP467.IPO_FRAME),$LOAD = SLOAD(FP467.TOOL_NO),$ACC = SACC_CP(LCPDAT467),$ORI_TYPE = SORI_TYP(LCPDAT467),$APO = SAPO(LCPDAT467),$JERK = SJERK(LCPDAT467),$COLLMON_TOL_PRO[1] = USE_CM_PRO_VALUES(0)
;ENDFOLD

;FOLD SLIN P468 Vel=1 m/s CPDAT468 Tool[4]:Microflown3D Base[2]:straight_sol;%{PE}
;FOLD Parameters ;%{h}
;Params IlfProvider=kukaroboter.basistech.inlineforms.movement.spline; Kuka.IsGlobalPoint=False; Kuka.PointName=P468; Kuka.BlendingEnabled=False; Kuka.MoveDataName=CPDAT468; Kuka.VelocityPath=1.000; Kuka.VelocityFieldEnabled=True; Kuka.ColDetectFieldEnabled=True; Kuka.CurrentCDSetIndex=0; Kuka.MovementParameterFieldEnabled=True; IlfCommand=SLIN
;ENDFOLD
SLIN XP468 WITH $VEL = SVEL_CP(2.0, , LCPDAT468),$TOOL = STOOL2(FP468),$BASE = SBASE(FP468.BASE_NO),$IPO_MODE = SIPO_MODE(FP468.IPO_FRAME),$LOAD = SLOAD(FP468.TOOL_NO),$ACC = SACC_CP(LCPDAT468),$ORI_TYPE = SORI_TYP(LCPDAT468),$APO = SAPO(LCPDAT468),$JERK = SJERK(LCPDAT468),$COLLMON_TOL_PRO[1] = USE_CM_PRO_VALUES(0)
;ENDFOLD

;FOLD SLIN P469 Vel=1 m/s CPDAT469 Tool[4]:Microflown3D Base[2]:straight_sol;%{PE}
;FOLD Parameters ;%{h}
;Params IlfProvider=kukaroboter.basistech.inlineforms.movement.spline; Kuka.IsGlobalPoint=False; Kuka.PointName=P469; Kuka.BlendingEnabled=False; Kuka.MoveDataName=CPDAT469; Kuka.VelocityPath=1.000; Kuka.VelocityFieldEnabled=True; Kuka.ColDetectFieldEnabled=True; Kuka.CurrentCDSetIndex=0; Kuka.MovementParameterFieldEnabled=True; IlfCommand=SLIN
;ENDFOLD
SLIN XP469 WITH $VEL = SVEL_CP(2.0, , LCPDAT469),$TOOL = STOOL2(FP469),$BASE = SBASE(FP469.BASE_NO),$IPO_MODE = SIPO_MODE(FP469.IPO_FRAME),$LOAD = SLOAD(FP469.TOOL_NO),$ACC = SACC_CP(LCPDAT469),$ORI_TYPE = SORI_TYP(LCPDAT469),$APO = SAPO(LCPDAT469),$JERK = SJERK(LCPDAT469),$COLLMON_TOL_PRO[1] = USE_CM_PRO_VALUES(0)
;ENDFOLD

;FOLD SLIN P470 Vel=1 m/s CPDAT470 Tool[4]:Microflown3D Base[2]:straight_sol;%{PE}
;FOLD Parameters ;%{h}
;Params IlfProvider=kukaroboter.basistech.inlineforms.movement.spline; Kuka.IsGlobalPoint=False; Kuka.PointName=P470; Kuka.BlendingEnabled=False; Kuka.MoveDataName=CPDAT470; Kuka.VelocityPath=1.000; Kuka.VelocityFieldEnabled=True; Kuka.ColDetectFieldEnabled=True; Kuka.CurrentCDSetIndex=0; Kuka.MovementParameterFieldEnabled=True; IlfCommand=SLIN
;ENDFOLD
SLIN XP470 WITH $VEL = SVEL_CP(2.0, , LCPDAT470),$TOOL = STOOL2(FP470),$BASE = SBASE(FP470.BASE_NO),$IPO_MODE = SIPO_MODE(FP470.IPO_FRAME),$LOAD = SLOAD(FP470.TOOL_NO),$ACC = SACC_CP(LCPDAT470),$ORI_TYPE = SORI_TYP(LCPDAT470),$APO = SAPO(LCPDAT470),$JERK = SJERK(LCPDAT470),$COLLMON_TOL_PRO[1] = USE_CM_PRO_VALUES(0)
;ENDFOLD

;FOLD SLIN P471 Vel=1 m/s CPDAT471 Tool[4]:Microflown3D Base[2]:straight_sol;%{PE}
;FOLD Parameters ;%{h}
;Params IlfProvider=kukaroboter.basistech.inlineforms.movement.spline; Kuka.IsGlobalPoint=False; Kuka.PointName=P471; Kuka.BlendingEnabled=False; Kuka.MoveDataName=CPDAT471; Kuka.VelocityPath=1.000; Kuka.VelocityFieldEnabled=True; Kuka.ColDetectFieldEnabled=True; Kuka.CurrentCDSetIndex=0; Kuka.MovementParameterFieldEnabled=True; IlfCommand=SLIN
;ENDFOLD
SLIN XP471 WITH $VEL = SVEL_CP(2.0, , LCPDAT471),$TOOL = STOOL2(FP471),$BASE = SBASE(FP471.BASE_NO),$IPO_MODE = SIPO_MODE(FP471.IPO_FRAME),$LOAD = SLOAD(FP471.TOOL_NO),$ACC = SACC_CP(LCPDAT471),$ORI_TYPE = SORI_TYP(LCPDAT471),$APO = SAPO(LCPDAT471),$JERK = SJERK(LCPDAT471),$COLLMON_TOL_PRO[1] = USE_CM_PRO_VALUES(0)
;ENDFOLD

;FOLD SLIN P472 Vel=1 m/s CPDAT472 Tool[4]:Microflown3D Base[2]:straight_sol;%{PE}
;FOLD Parameters ;%{h}
;Params IlfProvider=kukaroboter.basistech.inlineforms.movement.spline; Kuka.IsGlobalPoint=False; Kuka.PointName=P472; Kuka.BlendingEnabled=False; Kuka.MoveDataName=CPDAT472; Kuka.VelocityPath=1.000; Kuka.VelocityFieldEnabled=True; Kuka.ColDetectFieldEnabled=True; Kuka.CurrentCDSetIndex=0; Kuka.MovementParameterFieldEnabled=True; IlfCommand=SLIN
;ENDFOLD
SLIN XP472 WITH $VEL = SVEL_CP(2.0, , LCPDAT472),$TOOL = STOOL2(FP472),$BASE = SBASE(FP472.BASE_NO),$IPO_MODE = SIPO_MODE(FP472.IPO_FRAME),$LOAD = SLOAD(FP472.TOOL_NO),$ACC = SACC_CP(LCPDAT472),$ORI_TYPE = SORI_TYP(LCPDAT472),$APO = SAPO(LCPDAT472),$JERK = SJERK(LCPDAT472),$COLLMON_TOL_PRO[1] = USE_CM_PRO_VALUES(0)
;ENDFOLD

;FOLD SLIN P473 Vel=1 m/s CPDAT473 Tool[4]:Microflown3D Base[2]:straight_sol;%{PE}
;FOLD Parameters ;%{h}
;Params IlfProvider=kukaroboter.basistech.inlineforms.movement.spline; Kuka.IsGlobalPoint=False; Kuka.PointName=P473; Kuka.BlendingEnabled=False; Kuka.MoveDataName=CPDAT473; Kuka.VelocityPath=1.000; Kuka.VelocityFieldEnabled=True; Kuka.ColDetectFieldEnabled=True; Kuka.CurrentCDSetIndex=0; Kuka.MovementParameterFieldEnabled=True; IlfCommand=SLIN
;ENDFOLD
SLIN XP473 WITH $VEL = SVEL_CP(2.0, , LCPDAT473),$TOOL = STOOL2(FP473),$BASE = SBASE(FP473.BASE_NO),$IPO_MODE = SIPO_MODE(FP473.IPO_FRAME),$LOAD = SLOAD(FP473.TOOL_NO),$ACC = SACC_CP(LCPDAT473),$ORI_TYPE = SORI_TYP(LCPDAT473),$APO = SAPO(LCPDAT473),$JERK = SJERK(LCPDAT473),$COLLMON_TOL_PRO[1] = USE_CM_PRO_VALUES(0)
;ENDFOLD

;FOLD SLIN P474 Vel=1 m/s CPDAT474 Tool[4]:Microflown3D Base[2]:straight_sol;%{PE}
;FOLD Parameters ;%{h}
;Params IlfProvider=kukaroboter.basistech.inlineforms.movement.spline; Kuka.IsGlobalPoint=False; Kuka.PointName=P474; Kuka.BlendingEnabled=False; Kuka.MoveDataName=CPDAT474; Kuka.VelocityPath=1.000; Kuka.VelocityFieldEnabled=True; Kuka.ColDetectFieldEnabled=True; Kuka.CurrentCDSetIndex=0; Kuka.MovementParameterFieldEnabled=True; IlfCommand=SLIN
;ENDFOLD
SLIN XP474 WITH $VEL = SVEL_CP(2.0, , LCPDAT474),$TOOL = STOOL2(FP474),$BASE = SBASE(FP474.BASE_NO),$IPO_MODE = SIPO_MODE(FP474.IPO_FRAME),$LOAD = SLOAD(FP474.TOOL_NO),$ACC = SACC_CP(LCPDAT474),$ORI_TYPE = SORI_TYP(LCPDAT474),$APO = SAPO(LCPDAT474),$JERK = SJERK(LCPDAT474),$COLLMON_TOL_PRO[1] = USE_CM_PRO_VALUES(0)
;ENDFOLD

;FOLD SLIN P475 Vel=1 m/s CPDAT475 Tool[4]:Microflown3D Base[2]:straight_sol;%{PE}
;FOLD Parameters ;%{h}
;Params IlfProvider=kukaroboter.basistech.inlineforms.movement.spline; Kuka.IsGlobalPoint=False; Kuka.PointName=P475; Kuka.BlendingEnabled=False; Kuka.MoveDataName=CPDAT475; Kuka.VelocityPath=1.000; Kuka.VelocityFieldEnabled=True; Kuka.ColDetectFieldEnabled=True; Kuka.CurrentCDSetIndex=0; Kuka.MovementParameterFieldEnabled=True; IlfCommand=SLIN
;ENDFOLD
SLIN XP475 WITH $VEL = SVEL_CP(2.0, , LCPDAT475),$TOOL = STOOL2(FP475),$BASE = SBASE(FP475.BASE_NO),$IPO_MODE = SIPO_MODE(FP475.IPO_FRAME),$LOAD = SLOAD(FP475.TOOL_NO),$ACC = SACC_CP(LCPDAT475),$ORI_TYPE = SORI_TYP(LCPDAT475),$APO = SAPO(LCPDAT475),$JERK = SJERK(LCPDAT475),$COLLMON_TOL_PRO[1] = USE_CM_PRO_VALUES(0)
;ENDFOLD

;FOLD SLIN P476 Vel=1 m/s CPDAT476 Tool[4]:Microflown3D Base[2]:straight_sol;%{PE}
;FOLD Parameters ;%{h}
;Params IlfProvider=kukaroboter.basistech.inlineforms.movement.spline; Kuka.IsGlobalPoint=False; Kuka.PointName=P476; Kuka.BlendingEnabled=False; Kuka.MoveDataName=CPDAT476; Kuka.VelocityPath=1.000; Kuka.VelocityFieldEnabled=True; Kuka.ColDetectFieldEnabled=True; Kuka.CurrentCDSetIndex=0; Kuka.MovementParameterFieldEnabled=True; IlfCommand=SLIN
;ENDFOLD
SLIN XP476 WITH $VEL = SVEL_CP(2.0, , LCPDAT476),$TOOL = STOOL2(FP476),$BASE = SBASE(FP476.BASE_NO),$IPO_MODE = SIPO_MODE(FP476.IPO_FRAME),$LOAD = SLOAD(FP476.TOOL_NO),$ACC = SACC_CP(LCPDAT476),$ORI_TYPE = SORI_TYP(LCPDAT476),$APO = SAPO(LCPDAT476),$JERK = SJERK(LCPDAT476),$COLLMON_TOL_PRO[1] = USE_CM_PRO_VALUES(0)
;ENDFOLD

;FOLD SLIN P477 Vel=1 m/s CPDAT477 Tool[4]:Microflown3D Base[2]:straight_sol;%{PE}
;FOLD Parameters ;%{h}
;Params IlfProvider=kukaroboter.basistech.inlineforms.movement.spline; Kuka.IsGlobalPoint=False; Kuka.PointName=P477; Kuka.BlendingEnabled=False; Kuka.MoveDataName=CPDAT477; Kuka.VelocityPath=1.000; Kuka.VelocityFieldEnabled=True; Kuka.ColDetectFieldEnabled=True; Kuka.CurrentCDSetIndex=0; Kuka.MovementParameterFieldEnabled=True; IlfCommand=SLIN
;ENDFOLD
SLIN XP477 WITH $VEL = SVEL_CP(2.0, , LCPDAT477),$TOOL = STOOL2(FP477),$BASE = SBASE(FP477.BASE_NO),$IPO_MODE = SIPO_MODE(FP477.IPO_FRAME),$LOAD = SLOAD(FP477.TOOL_NO),$ACC = SACC_CP(LCPDAT477),$ORI_TYPE = SORI_TYP(LCPDAT477),$APO = SAPO(LCPDAT477),$JERK = SJERK(LCPDAT477),$COLLMON_TOL_PRO[1] = USE_CM_PRO_VALUES(0)
;ENDFOLD

;FOLD SLIN P478 Vel=1 m/s CPDAT478 Tool[4]:Microflown3D Base[2]:straight_sol;%{PE}
;FOLD Parameters ;%{h}
;Params IlfProvider=kukaroboter.basistech.inlineforms.movement.spline; Kuka.IsGlobalPoint=False; Kuka.PointName=P478; Kuka.BlendingEnabled=False; Kuka.MoveDataName=CPDAT478; Kuka.VelocityPath=1.000; Kuka.VelocityFieldEnabled=True; Kuka.ColDetectFieldEnabled=True; Kuka.CurrentCDSetIndex=0; Kuka.MovementParameterFieldEnabled=True; IlfCommand=SLIN
;ENDFOLD
SLIN XP478 WITH $VEL = SVEL_CP(2.0, , LCPDAT478),$TOOL = STOOL2(FP478),$BASE = SBASE(FP478.BASE_NO),$IPO_MODE = SIPO_MODE(FP478.IPO_FRAME),$LOAD = SLOAD(FP478.TOOL_NO),$ACC = SACC_CP(LCPDAT478),$ORI_TYPE = SORI_TYP(LCPDAT478),$APO = SAPO(LCPDAT478),$JERK = SJERK(LCPDAT478),$COLLMON_TOL_PRO[1] = USE_CM_PRO_VALUES(0)
;ENDFOLD

;FOLD SLIN P479 Vel=1 m/s CPDAT479 Tool[4]:Microflown3D Base[2]:straight_sol;%{PE}
;FOLD Parameters ;%{h}
;Params IlfProvider=kukaroboter.basistech.inlineforms.movement.spline; Kuka.IsGlobalPoint=False; Kuka.PointName=P479; Kuka.BlendingEnabled=False; Kuka.MoveDataName=CPDAT479; Kuka.VelocityPath=1.000; Kuka.VelocityFieldEnabled=True; Kuka.ColDetectFieldEnabled=True; Kuka.CurrentCDSetIndex=0; Kuka.MovementParameterFieldEnabled=True; IlfCommand=SLIN
;ENDFOLD
SLIN XP479 WITH $VEL = SVEL_CP(2.0, , LCPDAT479),$TOOL = STOOL2(FP479),$BASE = SBASE(FP479.BASE_NO),$IPO_MODE = SIPO_MODE(FP479.IPO_FRAME),$LOAD = SLOAD(FP479.TOOL_NO),$ACC = SACC_CP(LCPDAT479),$ORI_TYPE = SORI_TYP(LCPDAT479),$APO = SAPO(LCPDAT479),$JERK = SJERK(LCPDAT479),$COLLMON_TOL_PRO[1] = USE_CM_PRO_VALUES(0)
;ENDFOLD

;FOLD SLIN P480 Vel=1 m/s CPDAT480 Tool[4]:Microflown3D Base[2]:straight_sol;%{PE}
;FOLD Parameters ;%{h}
;Params IlfProvider=kukaroboter.basistech.inlineforms.movement.spline; Kuka.IsGlobalPoint=False; Kuka.PointName=P480; Kuka.BlendingEnabled=False; Kuka.MoveDataName=CPDAT480; Kuka.VelocityPath=1.000; Kuka.VelocityFieldEnabled=True; Kuka.ColDetectFieldEnabled=True; Kuka.CurrentCDSetIndex=0; Kuka.MovementParameterFieldEnabled=True; IlfCommand=SLIN
;ENDFOLD
SLIN XP480 WITH $VEL = SVEL_CP(2.0, , LCPDAT480),$TOOL = STOOL2(FP480),$BASE = SBASE(FP480.BASE_NO),$IPO_MODE = SIPO_MODE(FP480.IPO_FRAME),$LOAD = SLOAD(FP480.TOOL_NO),$ACC = SACC_CP(LCPDAT480),$ORI_TYPE = SORI_TYP(LCPDAT480),$APO = SAPO(LCPDAT480),$JERK = SJERK(LCPDAT480),$COLLMON_TOL_PRO[1] = USE_CM_PRO_VALUES(0)
;ENDFOLD

;FOLD SLIN P481 Vel=1 m/s CPDAT481 Tool[4]:Microflown3D Base[2]:straight_sol;%{PE}
;FOLD Parameters ;%{h}
;Params IlfProvider=kukaroboter.basistech.inlineforms.movement.spline; Kuka.IsGlobalPoint=False; Kuka.PointName=P481; Kuka.BlendingEnabled=False; Kuka.MoveDataName=CPDAT481; Kuka.VelocityPath=1.000; Kuka.VelocityFieldEnabled=True; Kuka.ColDetectFieldEnabled=True; Kuka.CurrentCDSetIndex=0; Kuka.MovementParameterFieldEnabled=True; IlfCommand=SLIN
;ENDFOLD
SLIN XP481 WITH $VEL = SVEL_CP(2.0, , LCPDAT481),$TOOL = STOOL2(FP481),$BASE = SBASE(FP481.BASE_NO),$IPO_MODE = SIPO_MODE(FP481.IPO_FRAME),$LOAD = SLOAD(FP481.TOOL_NO),$ACC = SACC_CP(LCPDAT481),$ORI_TYPE = SORI_TYP(LCPDAT481),$APO = SAPO(LCPDAT481),$JERK = SJERK(LCPDAT481),$COLLMON_TOL_PRO[1] = USE_CM_PRO_VALUES(0)
;ENDFOLD

;FOLD SLIN P482 Vel=1 m/s CPDAT482 Tool[4]:Microflown3D Base[2]:straight_sol;%{PE}
;FOLD Parameters ;%{h}
;Params IlfProvider=kukaroboter.basistech.inlineforms.movement.spline; Kuka.IsGlobalPoint=False; Kuka.PointName=P482; Kuka.BlendingEnabled=False; Kuka.MoveDataName=CPDAT482; Kuka.VelocityPath=1.000; Kuka.VelocityFieldEnabled=True; Kuka.ColDetectFieldEnabled=True; Kuka.CurrentCDSetIndex=0; Kuka.MovementParameterFieldEnabled=True; IlfCommand=SLIN
;ENDFOLD
SLIN XP482 WITH $VEL = SVEL_CP(2.0, , LCPDAT482),$TOOL = STOOL2(FP482),$BASE = SBASE(FP482.BASE_NO),$IPO_MODE = SIPO_MODE(FP482.IPO_FRAME),$LOAD = SLOAD(FP482.TOOL_NO),$ACC = SACC_CP(LCPDAT482),$ORI_TYPE = SORI_TYP(LCPDAT482),$APO = SAPO(LCPDAT482),$JERK = SJERK(LCPDAT482),$COLLMON_TOL_PRO[1] = USE_CM_PRO_VALUES(0)
;ENDFOLD

;FOLD SLIN P483 Vel=1 m/s CPDAT483 Tool[4]:Microflown3D Base[2]:straight_sol;%{PE}
;FOLD Parameters ;%{h}
;Params IlfProvider=kukaroboter.basistech.inlineforms.movement.spline; Kuka.IsGlobalPoint=False; Kuka.PointName=P483; Kuka.BlendingEnabled=False; Kuka.MoveDataName=CPDAT483; Kuka.VelocityPath=1.000; Kuka.VelocityFieldEnabled=True; Kuka.ColDetectFieldEnabled=True; Kuka.CurrentCDSetIndex=0; Kuka.MovementParameterFieldEnabled=True; IlfCommand=SLIN
;ENDFOLD
SLIN XP483 WITH $VEL = SVEL_CP(2.0, , LCPDAT483),$TOOL = STOOL2(FP483),$BASE = SBASE(FP483.BASE_NO),$IPO_MODE = SIPO_MODE(FP483.IPO_FRAME),$LOAD = SLOAD(FP483.TOOL_NO),$ACC = SACC_CP(LCPDAT483),$ORI_TYPE = SORI_TYP(LCPDAT483),$APO = SAPO(LCPDAT483),$JERK = SJERK(LCPDAT483),$COLLMON_TOL_PRO[1] = USE_CM_PRO_VALUES(0)
;ENDFOLD

;FOLD SLIN P484 Vel=1 m/s CPDAT484 Tool[4]:Microflown3D Base[2]:straight_sol;%{PE}
;FOLD Parameters ;%{h}
;Params IlfProvider=kukaroboter.basistech.inlineforms.movement.spline; Kuka.IsGlobalPoint=False; Kuka.PointName=P484; Kuka.BlendingEnabled=False; Kuka.MoveDataName=CPDAT484; Kuka.VelocityPath=1.000; Kuka.VelocityFieldEnabled=True; Kuka.ColDetectFieldEnabled=True; Kuka.CurrentCDSetIndex=0; Kuka.MovementParameterFieldEnabled=True; IlfCommand=SLIN
;ENDFOLD
SLIN XP484 WITH $VEL = SVEL_CP(2.0, , LCPDAT484),$TOOL = STOOL2(FP484),$BASE = SBASE(FP484.BASE_NO),$IPO_MODE = SIPO_MODE(FP484.IPO_FRAME),$LOAD = SLOAD(FP484.TOOL_NO),$ACC = SACC_CP(LCPDAT484),$ORI_TYPE = SORI_TYP(LCPDAT484),$APO = SAPO(LCPDAT484),$JERK = SJERK(LCPDAT484),$COLLMON_TOL_PRO[1] = USE_CM_PRO_VALUES(0)
;ENDFOLD

;FOLD SLIN P485 Vel=1 m/s CPDAT485 Tool[4]:Microflown3D Base[2]:straight_sol;%{PE}
;FOLD Parameters ;%{h}
;Params IlfProvider=kukaroboter.basistech.inlineforms.movement.spline; Kuka.IsGlobalPoint=False; Kuka.PointName=P485; Kuka.BlendingEnabled=False; Kuka.MoveDataName=CPDAT485; Kuka.VelocityPath=1.000; Kuka.VelocityFieldEnabled=True; Kuka.ColDetectFieldEnabled=True; Kuka.CurrentCDSetIndex=0; Kuka.MovementParameterFieldEnabled=True; IlfCommand=SLIN
;ENDFOLD
SLIN XP485 WITH $VEL = SVEL_CP(2.0, , LCPDAT485),$TOOL = STOOL2(FP485),$BASE = SBASE(FP485.BASE_NO),$IPO_MODE = SIPO_MODE(FP485.IPO_FRAME),$LOAD = SLOAD(FP485.TOOL_NO),$ACC = SACC_CP(LCPDAT485),$ORI_TYPE = SORI_TYP(LCPDAT485),$APO = SAPO(LCPDAT485),$JERK = SJERK(LCPDAT485),$COLLMON_TOL_PRO[1] = USE_CM_PRO_VALUES(0)
;ENDFOLD

;FOLD SLIN P486 Vel=1 m/s CPDAT486 Tool[4]:Microflown3D Base[2]:straight_sol;%{PE}
;FOLD Parameters ;%{h}
;Params IlfProvider=kukaroboter.basistech.inlineforms.movement.spline; Kuka.IsGlobalPoint=False; Kuka.PointName=P486; Kuka.BlendingEnabled=False; Kuka.MoveDataName=CPDAT486; Kuka.VelocityPath=1.000; Kuka.VelocityFieldEnabled=True; Kuka.ColDetectFieldEnabled=True; Kuka.CurrentCDSetIndex=0; Kuka.MovementParameterFieldEnabled=True; IlfCommand=SLIN
;ENDFOLD
SLIN XP486 WITH $VEL = SVEL_CP(2.0, , LCPDAT486),$TOOL = STOOL2(FP486),$BASE = SBASE(FP486.BASE_NO),$IPO_MODE = SIPO_MODE(FP486.IPO_FRAME),$LOAD = SLOAD(FP486.TOOL_NO),$ACC = SACC_CP(LCPDAT486),$ORI_TYPE = SORI_TYP(LCPDAT486),$APO = SAPO(LCPDAT486),$JERK = SJERK(LCPDAT486),$COLLMON_TOL_PRO[1] = USE_CM_PRO_VALUES(0)
;ENDFOLD

;FOLD SLIN P487 Vel=1 m/s CPDAT487 Tool[4]:Microflown3D Base[2]:straight_sol;%{PE}
;FOLD Parameters ;%{h}
;Params IlfProvider=kukaroboter.basistech.inlineforms.movement.spline; Kuka.IsGlobalPoint=False; Kuka.PointName=P487; Kuka.BlendingEnabled=False; Kuka.MoveDataName=CPDAT487; Kuka.VelocityPath=1.000; Kuka.VelocityFieldEnabled=True; Kuka.ColDetectFieldEnabled=True; Kuka.CurrentCDSetIndex=0; Kuka.MovementParameterFieldEnabled=True; IlfCommand=SLIN
;ENDFOLD
SLIN XP487 WITH $VEL = SVEL_CP(2.0, , LCPDAT487),$TOOL = STOOL2(FP487),$BASE = SBASE(FP487.BASE_NO),$IPO_MODE = SIPO_MODE(FP487.IPO_FRAME),$LOAD = SLOAD(FP487.TOOL_NO),$ACC = SACC_CP(LCPDAT487),$ORI_TYPE = SORI_TYP(LCPDAT487),$APO = SAPO(LCPDAT487),$JERK = SJERK(LCPDAT487),$COLLMON_TOL_PRO[1] = USE_CM_PRO_VALUES(0)
;ENDFOLD

;FOLD SLIN P488 Vel=1 m/s CPDAT488 Tool[4]:Microflown3D Base[2]:straight_sol;%{PE}
;FOLD Parameters ;%{h}
;Params IlfProvider=kukaroboter.basistech.inlineforms.movement.spline; Kuka.IsGlobalPoint=False; Kuka.PointName=P488; Kuka.BlendingEnabled=False; Kuka.MoveDataName=CPDAT488; Kuka.VelocityPath=1.000; Kuka.VelocityFieldEnabled=True; Kuka.ColDetectFieldEnabled=True; Kuka.CurrentCDSetIndex=0; Kuka.MovementParameterFieldEnabled=True; IlfCommand=SLIN
;ENDFOLD
SLIN XP488 WITH $VEL = SVEL_CP(2.0, , LCPDAT488),$TOOL = STOOL2(FP488),$BASE = SBASE(FP488.BASE_NO),$IPO_MODE = SIPO_MODE(FP488.IPO_FRAME),$LOAD = SLOAD(FP488.TOOL_NO),$ACC = SACC_CP(LCPDAT488),$ORI_TYPE = SORI_TYP(LCPDAT488),$APO = SAPO(LCPDAT488),$JERK = SJERK(LCPDAT488),$COLLMON_TOL_PRO[1] = USE_CM_PRO_VALUES(0)
;ENDFOLD

;FOLD SLIN P489 Vel=1 m/s CPDAT489 Tool[4]:Microflown3D Base[2]:straight_sol;%{PE}
;FOLD Parameters ;%{h}
;Params IlfProvider=kukaroboter.basistech.inlineforms.movement.spline; Kuka.IsGlobalPoint=False; Kuka.PointName=P489; Kuka.BlendingEnabled=False; Kuka.MoveDataName=CPDAT489; Kuka.VelocityPath=1.000; Kuka.VelocityFieldEnabled=True; Kuka.ColDetectFieldEnabled=True; Kuka.CurrentCDSetIndex=0; Kuka.MovementParameterFieldEnabled=True; IlfCommand=SLIN
;ENDFOLD
SLIN XP489 WITH $VEL = SVEL_CP(2.0, , LCPDAT489),$TOOL = STOOL2(FP489),$BASE = SBASE(FP489.BASE_NO),$IPO_MODE = SIPO_MODE(FP489.IPO_FRAME),$LOAD = SLOAD(FP489.TOOL_NO),$ACC = SACC_CP(LCPDAT489),$ORI_TYPE = SORI_TYP(LCPDAT489),$APO = SAPO(LCPDAT489),$JERK = SJERK(LCPDAT489),$COLLMON_TOL_PRO[1] = USE_CM_PRO_VALUES(0)
;ENDFOLD

;FOLD SLIN P490 Vel=1 m/s CPDAT490 Tool[4]:Microflown3D Base[2]:straight_sol;%{PE}
;FOLD Parameters ;%{h}
;Params IlfProvider=kukaroboter.basistech.inlineforms.movement.spline; Kuka.IsGlobalPoint=False; Kuka.PointName=P490; Kuka.BlendingEnabled=False; Kuka.MoveDataName=CPDAT490; Kuka.VelocityPath=1.000; Kuka.VelocityFieldEnabled=True; Kuka.ColDetectFieldEnabled=True; Kuka.CurrentCDSetIndex=0; Kuka.MovementParameterFieldEnabled=True; IlfCommand=SLIN
;ENDFOLD
SLIN XP490 WITH $VEL = SVEL_CP(2.0, , LCPDAT490),$TOOL = STOOL2(FP490),$BASE = SBASE(FP490.BASE_NO),$IPO_MODE = SIPO_MODE(FP490.IPO_FRAME),$LOAD = SLOAD(FP490.TOOL_NO),$ACC = SACC_CP(LCPDAT490),$ORI_TYPE = SORI_TYP(LCPDAT490),$APO = SAPO(LCPDAT490),$JERK = SJERK(LCPDAT490),$COLLMON_TOL_PRO[1] = USE_CM_PRO_VALUES(0)
;ENDFOLD

;FOLD SLIN P491 Vel=1 m/s CPDAT491 Tool[4]:Microflown3D Base[2]:straight_sol;%{PE}
;FOLD Parameters ;%{h}
;Params IlfProvider=kukaroboter.basistech.inlineforms.movement.spline; Kuka.IsGlobalPoint=False; Kuka.PointName=P491; Kuka.BlendingEnabled=False; Kuka.MoveDataName=CPDAT491; Kuka.VelocityPath=1.000; Kuka.VelocityFieldEnabled=True; Kuka.ColDetectFieldEnabled=True; Kuka.CurrentCDSetIndex=0; Kuka.MovementParameterFieldEnabled=True; IlfCommand=SLIN
;ENDFOLD
SLIN XP491 WITH $VEL = SVEL_CP(2.0, , LCPDAT491),$TOOL = STOOL2(FP491),$BASE = SBASE(FP491.BASE_NO),$IPO_MODE = SIPO_MODE(FP491.IPO_FRAME),$LOAD = SLOAD(FP491.TOOL_NO),$ACC = SACC_CP(LCPDAT491),$ORI_TYPE = SORI_TYP(LCPDAT491),$APO = SAPO(LCPDAT491),$JERK = SJERK(LCPDAT491),$COLLMON_TOL_PRO[1] = USE_CM_PRO_VALUES(0)
;ENDFOLD

;FOLD SLIN P492 Vel=1 m/s CPDAT492 Tool[4]:Microflown3D Base[2]:straight_sol;%{PE}
;FOLD Parameters ;%{h}
;Params IlfProvider=kukaroboter.basistech.inlineforms.movement.spline; Kuka.IsGlobalPoint=False; Kuka.PointName=P492; Kuka.BlendingEnabled=False; Kuka.MoveDataName=CPDAT492; Kuka.VelocityPath=1.000; Kuka.VelocityFieldEnabled=True; Kuka.ColDetectFieldEnabled=True; Kuka.CurrentCDSetIndex=0; Kuka.MovementParameterFieldEnabled=True; IlfCommand=SLIN
;ENDFOLD
SLIN XP492 WITH $VEL = SVEL_CP(2.0, , LCPDAT492),$TOOL = STOOL2(FP492),$BASE = SBASE(FP492.BASE_NO),$IPO_MODE = SIPO_MODE(FP492.IPO_FRAME),$LOAD = SLOAD(FP492.TOOL_NO),$ACC = SACC_CP(LCPDAT492),$ORI_TYPE = SORI_TYP(LCPDAT492),$APO = SAPO(LCPDAT492),$JERK = SJERK(LCPDAT492),$COLLMON_TOL_PRO[1] = USE_CM_PRO_VALUES(0)
;ENDFOLD

;FOLD SLIN P493 Vel=1 m/s CPDAT493 Tool[4]:Microflown3D Base[2]:straight_sol;%{PE}
;FOLD Parameters ;%{h}
;Params IlfProvider=kukaroboter.basistech.inlineforms.movement.spline; Kuka.IsGlobalPoint=False; Kuka.PointName=P493; Kuka.BlendingEnabled=False; Kuka.MoveDataName=CPDAT493; Kuka.VelocityPath=1.000; Kuka.VelocityFieldEnabled=True; Kuka.ColDetectFieldEnabled=True; Kuka.CurrentCDSetIndex=0; Kuka.MovementParameterFieldEnabled=True; IlfCommand=SLIN
;ENDFOLD
SLIN XP493 WITH $VEL = SVEL_CP(2.0, , LCPDAT493),$TOOL = STOOL2(FP493),$BASE = SBASE(FP493.BASE_NO),$IPO_MODE = SIPO_MODE(FP493.IPO_FRAME),$LOAD = SLOAD(FP493.TOOL_NO),$ACC = SACC_CP(LCPDAT493),$ORI_TYPE = SORI_TYP(LCPDAT493),$APO = SAPO(LCPDAT493),$JERK = SJERK(LCPDAT493),$COLLMON_TOL_PRO[1] = USE_CM_PRO_VALUES(0)
;ENDFOLD

;FOLD SLIN P494 Vel=1 m/s CPDAT494 Tool[4]:Microflown3D Base[2]:straight_sol;%{PE}
;FOLD Parameters ;%{h}
;Params IlfProvider=kukaroboter.basistech.inlineforms.movement.spline; Kuka.IsGlobalPoint=False; Kuka.PointName=P494; Kuka.BlendingEnabled=False; Kuka.MoveDataName=CPDAT494; Kuka.VelocityPath=1.000; Kuka.VelocityFieldEnabled=True; Kuka.ColDetectFieldEnabled=True; Kuka.CurrentCDSetIndex=0; Kuka.MovementParameterFieldEnabled=True; IlfCommand=SLIN
;ENDFOLD
SLIN XP494 WITH $VEL = SVEL_CP(2.0, , LCPDAT494),$TOOL = STOOL2(FP494),$BASE = SBASE(FP494.BASE_NO),$IPO_MODE = SIPO_MODE(FP494.IPO_FRAME),$LOAD = SLOAD(FP494.TOOL_NO),$ACC = SACC_CP(LCPDAT494),$ORI_TYPE = SORI_TYP(LCPDAT494),$APO = SAPO(LCPDAT494),$JERK = SJERK(LCPDAT494),$COLLMON_TOL_PRO[1] = USE_CM_PRO_VALUES(0)
;ENDFOLD

;FOLD SLIN P495 Vel=1 m/s CPDAT495 Tool[4]:Microflown3D Base[2]:straight_sol;%{PE}
;FOLD Parameters ;%{h}
;Params IlfProvider=kukaroboter.basistech.inlineforms.movement.spline; Kuka.IsGlobalPoint=False; Kuka.PointName=P495; Kuka.BlendingEnabled=False; Kuka.MoveDataName=CPDAT495; Kuka.VelocityPath=1.000; Kuka.VelocityFieldEnabled=True; Kuka.ColDetectFieldEnabled=True; Kuka.CurrentCDSetIndex=0; Kuka.MovementParameterFieldEnabled=True; IlfCommand=SLIN
;ENDFOLD
SLIN XP495 WITH $VEL = SVEL_CP(2.0, , LCPDAT495),$TOOL = STOOL2(FP495),$BASE = SBASE(FP495.BASE_NO),$IPO_MODE = SIPO_MODE(FP495.IPO_FRAME),$LOAD = SLOAD(FP495.TOOL_NO),$ACC = SACC_CP(LCPDAT495),$ORI_TYPE = SORI_TYP(LCPDAT495),$APO = SAPO(LCPDAT495),$JERK = SJERK(LCPDAT495),$COLLMON_TOL_PRO[1] = USE_CM_PRO_VALUES(0)
;ENDFOLD

;FOLD SLIN P496 Vel=1 m/s CPDAT496 Tool[4]:Microflown3D Base[2]:straight_sol;%{PE}
;FOLD Parameters ;%{h}
;Params IlfProvider=kukaroboter.basistech.inlineforms.movement.spline; Kuka.IsGlobalPoint=False; Kuka.PointName=P496; Kuka.BlendingEnabled=False; Kuka.MoveDataName=CPDAT496; Kuka.VelocityPath=1.000; Kuka.VelocityFieldEnabled=True; Kuka.ColDetectFieldEnabled=True; Kuka.CurrentCDSetIndex=0; Kuka.MovementParameterFieldEnabled=True; IlfCommand=SLIN
;ENDFOLD
SLIN XP496 WITH $VEL = SVEL_CP(2.0, , LCPDAT496),$TOOL = STOOL2(FP496),$BASE = SBASE(FP496.BASE_NO),$IPO_MODE = SIPO_MODE(FP496.IPO_FRAME),$LOAD = SLOAD(FP496.TOOL_NO),$ACC = SACC_CP(LCPDAT496),$ORI_TYPE = SORI_TYP(LCPDAT496),$APO = SAPO(LCPDAT496),$JERK = SJERK(LCPDAT496),$COLLMON_TOL_PRO[1] = USE_CM_PRO_VALUES(0)
;ENDFOLD

;FOLD SLIN P497 Vel=1 m/s CPDAT497 Tool[4]:Microflown3D Base[2]:straight_sol;%{PE}
;FOLD Parameters ;%{h}
;Params IlfProvider=kukaroboter.basistech.inlineforms.movement.spline; Kuka.IsGlobalPoint=False; Kuka.PointName=P497; Kuka.BlendingEnabled=False; Kuka.MoveDataName=CPDAT497; Kuka.VelocityPath=1.000; Kuka.VelocityFieldEnabled=True; Kuka.ColDetectFieldEnabled=True; Kuka.CurrentCDSetIndex=0; Kuka.MovementParameterFieldEnabled=True; IlfCommand=SLIN
;ENDFOLD
SLIN XP497 WITH $VEL = SVEL_CP(2.0, , LCPDAT497),$TOOL = STOOL2(FP497),$BASE = SBASE(FP497.BASE_NO),$IPO_MODE = SIPO_MODE(FP497.IPO_FRAME),$LOAD = SLOAD(FP497.TOOL_NO),$ACC = SACC_CP(LCPDAT497),$ORI_TYPE = SORI_TYP(LCPDAT497),$APO = SAPO(LCPDAT497),$JERK = SJERK(LCPDAT497),$COLLMON_TOL_PRO[1] = USE_CM_PRO_VALUES(0)
;ENDFOLD

;FOLD SLIN P498 Vel=1 m/s CPDAT498 Tool[4]:Microflown3D Base[2]:straight_sol;%{PE}
;FOLD Parameters ;%{h}
;Params IlfProvider=kukaroboter.basistech.inlineforms.movement.spline; Kuka.IsGlobalPoint=False; Kuka.PointName=P498; Kuka.BlendingEnabled=False; Kuka.MoveDataName=CPDAT498; Kuka.VelocityPath=1.000; Kuka.VelocityFieldEnabled=True; Kuka.ColDetectFieldEnabled=True; Kuka.CurrentCDSetIndex=0; Kuka.MovementParameterFieldEnabled=True; IlfCommand=SLIN
;ENDFOLD
SLIN XP498 WITH $VEL = SVEL_CP(2.0, , LCPDAT498),$TOOL = STOOL2(FP498),$BASE = SBASE(FP498.BASE_NO),$IPO_MODE = SIPO_MODE(FP498.IPO_FRAME),$LOAD = SLOAD(FP498.TOOL_NO),$ACC = SACC_CP(LCPDAT498),$ORI_TYPE = SORI_TYP(LCPDAT498),$APO = SAPO(LCPDAT498),$JERK = SJERK(LCPDAT498),$COLLMON_TOL_PRO[1] = USE_CM_PRO_VALUES(0)
;ENDFOLD

;FOLD SLIN P499 Vel=1 m/s CPDAT499 Tool[4]:Microflown3D Base[2]:straight_sol;%{PE}
;FOLD Parameters ;%{h}
;Params IlfProvider=kukaroboter.basistech.inlineforms.movement.spline; Kuka.IsGlobalPoint=False; Kuka.PointName=P499; Kuka.BlendingEnabled=False; Kuka.MoveDataName=CPDAT499; Kuka.VelocityPath=1.000; Kuka.VelocityFieldEnabled=True; Kuka.ColDetectFieldEnabled=True; Kuka.CurrentCDSetIndex=0; Kuka.MovementParameterFieldEnabled=True; IlfCommand=SLIN
;ENDFOLD
SLIN XP499 WITH $VEL = SVEL_CP(2.0, , LCPDAT499),$TOOL = STOOL2(FP499),$BASE = SBASE(FP499.BASE_NO),$IPO_MODE = SIPO_MODE(FP499.IPO_FRAME),$LOAD = SLOAD(FP499.TOOL_NO),$ACC = SACC_CP(LCPDAT499),$ORI_TYPE = SORI_TYP(LCPDAT499),$APO = SAPO(LCPDAT499),$JERK = SJERK(LCPDAT499),$COLLMON_TOL_PRO[1] = USE_CM_PRO_VALUES(0)
;ENDFOLD

;FOLD SLIN P500 Vel=1 m/s CPDAT500 Tool[4]:Microflown3D Base[2]:straight_sol;%{PE}
;FOLD Parameters ;%{h}
;Params IlfProvider=kukaroboter.basistech.inlineforms.movement.spline; Kuka.IsGlobalPoint=False; Kuka.PointName=P500; Kuka.BlendingEnabled=False; Kuka.MoveDataName=CPDAT500; Kuka.VelocityPath=1.000; Kuka.VelocityFieldEnabled=True; Kuka.ColDetectFieldEnabled=True; Kuka.CurrentCDSetIndex=0; Kuka.MovementParameterFieldEnabled=True; IlfCommand=SLIN
;ENDFOLD
SLIN XP500 WITH $VEL = SVEL_CP(2.0, , LCPDAT500),$TOOL = STOOL2(FP500),$BASE = SBASE(FP500.BASE_NO),$IPO_MODE = SIPO_MODE(FP500.IPO_FRAME),$LOAD = SLOAD(FP500.TOOL_NO),$ACC = SACC_CP(LCPDAT500),$ORI_TYPE = SORI_TYP(LCPDAT500),$APO = SAPO(LCPDAT500),$JERK = SJERK(LCPDAT500),$COLLMON_TOL_PRO[1] = USE_CM_PRO_VALUES(0)
;ENDFOLD

;FOLD SLIN P501 Vel=1 m/s CPDAT501 Tool[4]:Microflown3D Base[2]:straight_sol;%{PE}
;FOLD Parameters ;%{h}
;Params IlfProvider=kukaroboter.basistech.inlineforms.movement.spline; Kuka.IsGlobalPoint=False; Kuka.PointName=P501; Kuka.BlendingEnabled=False; Kuka.MoveDataName=CPDAT501; Kuka.VelocityPath=1.000; Kuka.VelocityFieldEnabled=True; Kuka.ColDetectFieldEnabled=True; Kuka.CurrentCDSetIndex=0; Kuka.MovementParameterFieldEnabled=True; IlfCommand=SLIN
;ENDFOLD
SLIN XP501 WITH $VEL = SVEL_CP(2.0, , LCPDAT501),$TOOL = STOOL2(FP501),$BASE = SBASE(FP501.BASE_NO),$IPO_MODE = SIPO_MODE(FP501.IPO_FRAME),$LOAD = SLOAD(FP501.TOOL_NO),$ACC = SACC_CP(LCPDAT501),$ORI_TYPE = SORI_TYP(LCPDAT501),$APO = SAPO(LCPDAT501),$JERK = SJERK(LCPDAT501),$COLLMON_TOL_PRO[1] = USE_CM_PRO_VALUES(0)
;ENDFOLD

;FOLD SLIN P502 Vel=1 m/s CPDAT502 Tool[4]:Microflown3D Base[2]:straight_sol;%{PE}
;FOLD Parameters ;%{h}
;Params IlfProvider=kukaroboter.basistech.inlineforms.movement.spline; Kuka.IsGlobalPoint=False; Kuka.PointName=P502; Kuka.BlendingEnabled=False; Kuka.MoveDataName=CPDAT502; Kuka.VelocityPath=1.000; Kuka.VelocityFieldEnabled=True; Kuka.ColDetectFieldEnabled=True; Kuka.CurrentCDSetIndex=0; Kuka.MovementParameterFieldEnabled=True; IlfCommand=SLIN
;ENDFOLD
SLIN XP502 WITH $VEL = SVEL_CP(2.0, , LCPDAT502),$TOOL = STOOL2(FP502),$BASE = SBASE(FP502.BASE_NO),$IPO_MODE = SIPO_MODE(FP502.IPO_FRAME),$LOAD = SLOAD(FP502.TOOL_NO),$ACC = SACC_CP(LCPDAT502),$ORI_TYPE = SORI_TYP(LCPDAT502),$APO = SAPO(LCPDAT502),$JERK = SJERK(LCPDAT502),$COLLMON_TOL_PRO[1] = USE_CM_PRO_VALUES(0)
;ENDFOLD

;FOLD SLIN P503 Vel=1 m/s CPDAT503 Tool[4]:Microflown3D Base[2]:straight_sol;%{PE}
;FOLD Parameters ;%{h}
;Params IlfProvider=kukaroboter.basistech.inlineforms.movement.spline; Kuka.IsGlobalPoint=False; Kuka.PointName=P503; Kuka.BlendingEnabled=False; Kuka.MoveDataName=CPDAT503; Kuka.VelocityPath=1.000; Kuka.VelocityFieldEnabled=True; Kuka.ColDetectFieldEnabled=True; Kuka.CurrentCDSetIndex=0; Kuka.MovementParameterFieldEnabled=True; IlfCommand=SLIN
;ENDFOLD
SLIN XP503 WITH $VEL = SVEL_CP(2.0, , LCPDAT503),$TOOL = STOOL2(FP503),$BASE = SBASE(FP503.BASE_NO),$IPO_MODE = SIPO_MODE(FP503.IPO_FRAME),$LOAD = SLOAD(FP503.TOOL_NO),$ACC = SACC_CP(LCPDAT503),$ORI_TYPE = SORI_TYP(LCPDAT503),$APO = SAPO(LCPDAT503),$JERK = SJERK(LCPDAT503),$COLLMON_TOL_PRO[1] = USE_CM_PRO_VALUES(0)
;ENDFOLD

;FOLD SLIN P504 Vel=1 m/s CPDAT504 Tool[4]:Microflown3D Base[2]:straight_sol;%{PE}
;FOLD Parameters ;%{h}
;Params IlfProvider=kukaroboter.basistech.inlineforms.movement.spline; Kuka.IsGlobalPoint=False; Kuka.PointName=P504; Kuka.BlendingEnabled=False; Kuka.MoveDataName=CPDAT504; Kuka.VelocityPath=1.000; Kuka.VelocityFieldEnabled=True; Kuka.ColDetectFieldEnabled=True; Kuka.CurrentCDSetIndex=0; Kuka.MovementParameterFieldEnabled=True; IlfCommand=SLIN
;ENDFOLD
SLIN XP504 WITH $VEL = SVEL_CP(2.0, , LCPDAT504),$TOOL = STOOL2(FP504),$BASE = SBASE(FP504.BASE_NO),$IPO_MODE = SIPO_MODE(FP504.IPO_FRAME),$LOAD = SLOAD(FP504.TOOL_NO),$ACC = SACC_CP(LCPDAT504),$ORI_TYPE = SORI_TYP(LCPDAT504),$APO = SAPO(LCPDAT504),$JERK = SJERK(LCPDAT504),$COLLMON_TOL_PRO[1] = USE_CM_PRO_VALUES(0)
;ENDFOLD

